LIN {X -0.176,Y -701.742,Z 1215.429,A 0.000,B 0.000,C 90.000,E1 113.259} C_DIS
LIN {X -0.039,Y -700.692,Z 1215.429,A 0.000,B 0.000,C 90.000,E1 113.131} C_DIS
LIN {X -0.019,Y -695.221,Z 1215.426,A 0.000,B 0.000,C 90.000,E1 112.695} C_DIS
LIN {X 0.002,Y -693.496,Z 1215.426,A 0.000,B 0.000,C 90.000,E1 112.589} C_DIS
LIN {X 0.017,Y -688.158,Z 1215.425,A 0.000,B 0.000,C 90.000,E1 112.408} C_DIS
LIN {X 0.322,Y -686.600,Z 1215.424,A 0.000,B 0.000,C 90.000,E1 112.333} C_DIS
LIN {X -0.036,Y -685.254,Z 1215.424,A 0.000,B 0.000,C 90.000,E1 112.333} C_DIS
LIN {X 0.238,Y -679.829,Z 1215.424,A 0.000,B 0.000,C 90.000,E1 112.280} C_DIS
LIN {X 0.132,Y -677.657,Z 1215.424,A 0.000,B 0.000,C 90.000,E1 112.280} C_DIS
LIN {X 0.079,Y -611.887,Z 1215.424,A 0.000,B 0.000,C 90.000,E1 112.280} C_DIS
LIN {X -0.103,Y -610.037,Z 1215.423,A 0.000,B 0.000,C 90.000,E1 112.206} C_DIS
LIN {X 0.141,Y -604.449,Z 1215.421,A 0.000,B 0.000,C 90.000,E1 111.791} C_DIS
LIN {X 0.099,Y -601.562,Z 1215.420,A 0.000,B 0.000,C 90.000,E1 111.535} C_DIS
LIN {X 0.143,Y -599.778,Z 1215.418,A 0.000,B 0.000,C 90.000,E1 111.280} C_DIS
LIN {X -0.112,Y -598.457,Z 1215.417,A 0.000,B 0.000,C 90.000,E1 111.153} C_DIS
LIN {X -0.155,Y -598.430,Z 1215.417,A 0.000,B 0.000,C 90.000,E1 111.153} C_DIS
LIN {X -0.070,Y -597.952,Z 1215.417,A 0.000,B 0.000,C 90.000,E1 110.972} C_DIS
LIN {X 0.221,Y -598.845,Z 1215.414,A 0.000,B 0.000,C 90.000,E1 110.482} C_DIS
LIN {X 0.094,Y -601.655,Z 1215.410,A 0.000,B 0.000,C 90.000,E1 109.704} C_DIS
LIN {X 0.200,Y -604.148,Z 1215.405,A 0.000,B 0.000,C 90.000,E1 108.906} C_DIS
LIN {X -0.243,Y -610.599,Z 1215.394,A 0.000,B 0.000,C 90.000,E1 106.858} C_DIS
LIN {X 0.087,Y -611.302,Z 1215.392,A 0.000,B 0.000,C 90.000,E1 106.567} C_DIS
LIN {X 0.007,Y -612.225,Z 1215.391,A 0.000,B 0.000,C 90.000,E1 106.315} C_DIS
LIN {X -0.145,Y -614.498,Z 1215.386,A 0.000,B 0.000,C 90.000,E1 105.552} C_DIS
LIN {X -0.108,Y -616.200,Z 1215.382,A 0.000,B 0.000,C 90.000,E1 104.773} C_DIS
LIN {X 0.020,Y -617.147,Z 1215.379,A 0.000,B 0.000,C 90.000,E1 104.245} C_DIS
LIN {X 0.159,Y -617.816,Z 1215.376,A 0.000,B 0.000,C 90.000,E1 103.716} C_DIS
LIN {X -0.157,Y -618.203,Z 1215.373,A 0.000,B 0.000,C 90.000,E1 103.231} C_DIS
LIN {X -0.014,Y -618.268,Z 1215.371,A 0.000,B 0.000,C 90.000,E1 102.703} C_DIS
LIN {X 0.360,Y -618.212,Z 1215.369,A 0.000,B 0.000,C 90.000,E1 102.411} C_DIS
LIN {X -0.229,Y -617.696,Z 1215.366,A 0.000,B 0.000,C 90.000,E1 101.951} C_DIS
LIN {X -0.083,Y -616.795,Z 1215.363,A 0.000,B 0.000,C 90.000,E1 101.422} C_DIS
LIN {X 0.054,Y -615.559,Z 1215.361,A 0.000,B 0.000,C 90.000,E1 100.894} C_DIS
LIN {X -0.184,Y -614.849,Z 1215.359,A 0.000,B 0.000,C 90.000,E1 100.658} C_DIS
LIN {X -0.172,Y -613.051,Z 1215.356,A 0.000,B 0.000,C 90.000,E1 100.141} C_DIS
LIN {X -0.242,Y -609.874,Z 1215.353,A 0.000,B 0.000,C 90.000,E1 99.500} C_DIS
LIN {X -0.077,Y -607.729,Z 1215.351,A 0.000,B 0.000,C 90.000,E1 99.095} C_DIS
LIN {X -0.198,Y -603.306,Z 1215.347,A 0.000,B 0.000,C 90.000,E1 98.454} C_DIS
LIN {X -0.254,Y -599.077,Z 1215.344,A 0.000,B 0.000,C 90.000,E1 97.936} C_DIS
LIN {X -0.212,Y -594.199,Z 1215.341,A 0.000,B 0.000,C 90.000,E1 97.409} C_DIS
LIN {X -0.018,Y -588.778,Z 1215.338,A 0.000,B 0.000,C 90.000,E1 96.891} C_DIS
LIN {X -0.118,Y -584.273,Z 1215.336,A 0.000,B 0.000,C 90.000,E1 96.543} C_DIS
LIN {X -0.046,Y -581.409,Z 1215.335,A 0.000,B 0.000,C 90.000,E1 96.315} C_DIS
LIN {X -0.022,Y -579.787,Z 1215.334,A 0.000,B 0.000,C 90.000,E1 96.201} C_DIS
LIN {X -0.082,Y -574.622,Z 1215.333,A 0.000,B 0.000,C 90.000,E1 95.910} C_DIS
LIN {X -0.113,Y -567.317,Z 1215.330,A 0.000,B 0.000,C 90.000,E1 95.454} C_DIS
LIN {X 0.093,Y -566.335,Z 1215.330,A 0.000,B 0.000,C 90.000,E1 95.334} C_DIS
LIN {X -0.087,Y -565.372,Z 1215.329,A 0.000,B 0.000,C 90.000,E1 95.220} C_DIS
LIN {X 0.152,Y -564.026,Z 1215.328,A 0.000,B 0.000,C 90.000,E1 94.935} C_DIS
LIN {X 0.109,Y -564.023,Z 1215.328,A 0.000,B 0.000,C 90.000,E1 94.935} C_DIS
LIN {X -0.143,Y -563.804,Z 1215.325,A 0.000,B 0.000,C 90.000,E1 94.531} C_DIS
LIN {X 0.187,Y -563.579,Z 1215.324,A 0.000,B 0.000,C 90.000,E1 94.359} C_DIS
LIN {X -0.278,Y -563.705,Z 1215.320,A 0.000,B 0.000,C 90.000,E1 93.555} C_DIS
LIN {X 0.274,Y -564.650,Z 1215.312,A 0.000,B 0.000,C 90.000,E1 92.121} C_DIS
LIN {X -0.062,Y -565.996,Z 1215.301,A 0.000,B 0.000,C 90.000,E1 90.229} C_DIS
LIN {X 0.068,Y -567.159,Z 1215.292,A 0.000,B 0.000,C 90.000,E1 88.568} C_DIS
LIN {X -0.007,Y -568.004,Z 1215.286,A 0.000,B 0.000,C 90.000,E1 87.478} C_DIS
LIN {X 0.210,Y -569.246,Z 1215.277,A 0.000,B 0.000,C 90.000,E1 85.812} C_DIS
LIN {X 0.060,Y -570.822,Z 1215.266,A 0.000,B 0.000,C 90.000,E1 83.913} C_DIS
LIN {X 0.201,Y -572.005,Z 1215.259,A 0.000,B 0.000,C 90.000,E1 82.534} C_DIS
LIN {X -0.060,Y -573.113,Z 1215.251,A 0.000,B 0.000,C 90.000,E1 81.197} C_DIS
LIN {X 0.274,Y -574.095,Z 1215.244,A 0.000,B 0.000,C 90.000,E1 79.803} C_DIS
LIN {X 0.259,Y -575.130,Z 1215.234,A 0.000,B 0.000,C 90.000,E1 78.173} C_DIS
LIN {X -0.189,Y -576.095,Z 1215.225,A 0.000,B 0.000,C 90.000,E1 76.589} C_DIS
LIN {X -0.132,Y -576.812,Z 1215.218,A 0.000,B 0.000,C 90.000,E1 75.227} C_DIS
LIN {X 0.303,Y -577.663,Z 1215.209,A 0.000,B 0.000,C 90.000,E1 73.559} C_DIS
LIN {X 0.223,Y -578.855,Z 1215.197,A 0.000,B 0.000,C 90.000,E1 71.402} C_DIS
LIN {X 0.002,Y -580.238,Z 1215.185,A 0.000,B 0.000,C 90.000,E1 69.263} C_DIS
LIN {X 0.067,Y -582.374,Z 1215.170,A 0.000,B 0.000,C 90.000,E1 66.561} C_DIS
LIN {X -0.194,Y -583.878,Z 1215.161,A 0.000,B 0.000,C 90.000,E1 64.973} C_DIS
LIN {X -0.014,Y -585.587,Z 1215.151,A 0.000,B 0.000,C 90.000,E1 63.076} C_DIS
LIN {X 0.054,Y -587.260,Z 1215.141,A 0.000,B 0.000,C 90.000,E1 61.463} C_DIS
LIN {X -0.073,Y -588.926,Z 1215.133,A 0.000,B 0.000,C 90.000,E1 59.871} C_DIS
LIN {X 0.147,Y -590.389,Z 1215.124,A 0.000,B 0.000,C 90.000,E1 58.250} C_DIS
LIN {X -0.005,Y -591.370,Z 1215.118,A 0.000,B 0.000,C 90.000,E1 57.199} C_DIS
LIN {X -0.002,Y -592.248,Z 1215.112,A 0.000,B 0.000,C 90.000,E1 56.135} C_DIS
LIN {X -0.218,Y -593.486,Z 1215.103,A 0.000,B 0.000,C 90.000,E1 54.562} C_DIS
LIN {X 0.269,Y -594.706,Z 1215.094,A 0.000,B 0.000,C 90.000,E1 52.924} C_DIS
LIN {X -0.141,Y -595.494,Z 1215.088,A 0.000,B 0.000,C 90.000,E1 51.904} C_DIS
LIN {X 0.290,Y -596.524,Z 1215.079,A 0.000,B 0.000,C 90.000,E1 50.275} C_DIS
LIN {X 0.285,Y -597.211,Z 1215.071,A 0.000,B 0.000,C 90.000,E1 48.690} C_DIS
LIN {X 0.064,Y -597.686,Z 1215.063,A 0.000,B 0.000,C 90.000,E1 47.391} C_DIS
LIN {X -0.156,Y -597.920,Z 1215.059,A 0.000,B 0.000,C 90.000,E1 46.620} C_DIS
LIN {X -0.179,Y -598.105,Z 1215.053,A 0.000,B 0.000,C 90.000,E1 45.567} C_DIS
LIN {X 0.019,Y -598.095,Z 1215.049,A 0.000,B 0.000,C 90.000,E1 44.757} C_DIS
LIN {X 0.217,Y -597.954,Z 1215.044,A 0.000,B 0.000,C 90.000,E1 43.947} C_DIS
LIN {X -0.217,Y -597.831,Z 1215.041,A 0.000,B 0.000,C 90.000,E1 43.461} C_DIS
LIN {X 0.186,Y -596.976,Z 1215.033,A 0.000,B 0.000,C 90.000,E1 41.838} C_DIS
LIN {X -0.040,Y -596.562,Z 1215.028,A 0.000,B 0.000,C 90.000,E1 41.067} C_DIS
LIN {X 0.175,Y -595.674,Z 1215.021,A 0.000,B 0.000,C 90.000,E1 39.725} C_DIS
LIN {X -0.072,Y -595.061,Z 1215.016,A 0.000,B 0.000,C 90.000,E1 38.955} C_DIS
LIN {X 0.208,Y -593.806,Z 1215.009,A 0.000,B 0.000,C 90.000,E1 37.604} C_DIS
LIN {X -0.216,Y -592.497,Z 1215.003,A 0.000,B 0.000,C 90.000,E1 36.583} C_DIS
LIN {X 0.215,Y -591.801,Z 1215.000,A 0.000,B 0.000,C 90.000,E1 36.011} C_DIS
LIN {X 0.100,Y -589.562,Z 1214.993,A 0.000,B 0.000,C 90.000,E1 34.692} C_DIS
LIN {X -0.115,Y -587.851,Z 1214.988,A 0.000,B 0.000,C 90.000,E1 33.913} C_DIS
LIN {X 0.138,Y -585.969,Z 1214.984,A 0.000,B 0.000,C 90.000,E1 33.086} C_DIS
LIN {X 0.187,Y -584.455,Z 1214.981,A 0.000,B 0.000,C 90.000,E1 32.546} C_DIS
LIN {X 0.258,Y -581.148,Z 1214.975,A 0.000,B 0.000,C 90.000,E1 31.465} C_DIS
LIN {X 0.130,Y -578.136,Z 1214.970,A 0.000,B 0.000,C 90.000,E1 30.669} C_DIS
LIN {X -0.016,Y -577.087,Z 1214.969,A 0.000,B 0.000,C 90.000,E1 30.413} C_DIS
LIN {X 0.024,Y -572.873,Z 1214.964,A 0.000,B 0.000,C 90.000,E1 29.461} C_DIS
LIN {X -0.303,Y -570.192,Z 1214.961,A 0.000,B 0.000,C 90.000,E1 28.949} C_DIS
LIN {X 0.215,Y -568.064,Z 1214.958,A 0.000,B 0.000,C 90.000,E1 28.487} C_DIS
LIN {X -0.231,Y -564.211,Z 1214.955,A 0.000,B 0.000,C 90.000,E1 27.847} C_DIS
LIN {X 0.151,Y -560.907,Z 1214.952,A 0.000,B 0.000,C 90.000,E1 27.257} C_DIS
LIN {X 0.045,Y -555.675,Z 1214.947,A 0.000,B 0.000,C 90.000,E1 26.437} C_DIS
LIN {X 0.242,Y -550.798,Z 1214.943,A 0.000,B 0.000,C 90.000,E1 25.720} C_DIS
LIN {X -0.221,Y -546.679,Z 1214.940,A 0.000,B 0.000,C 90.000,E1 25.207} C_DIS
LIN {X 0.149,Y -541.009,Z 1214.936,A 0.000,B 0.000,C 90.000,E1 24.463} C_DIS
LIN {X -0.020,Y -535.070,Z 1214.932,A 0.000,B 0.000,C 90.000,E1 23.770} C_DIS
LIN {X 0.160,Y -527.403,Z 1214.927,A 0.000,B 0.000,C 90.000,E1 22.898} C_DIS
LIN {X 0.124,Y -522.134,Z 1214.924,A 0.000,B 0.000,C 90.000,E1 22.333} C_DIS
LIN {X -0.185,Y -514.110,Z 1214.920,A 0.000,B 0.000,C 90.000,E1 21.535} C_DIS
LIN {X -0.222,Y -506.137,Z 1214.915,A 0.000,B 0.000,C 90.000,E1 20.737} C_DIS
LIN {X -0.144,Y -499.081,Z 1214.911,A 0.000,B 0.000,C 90.000,E1 20.047} C_DIS
LIN {X -0.219,Y -490.622,Z 1214.907,A 0.000,B 0.000,C 90.000,E1 19.268} C_DIS
LIN {X -0.006,Y -484.930,Z 1214.904,A 0.000,B 0.000,C 90.000,E1 18.725} C_DIS
LIN {X -0.059,Y -474.720,Z 1214.899,A 0.000,B 0.000,C 90.000,E1 17.819} C_DIS
LIN {X 0.239,Y -460.231,Z 1214.892,A 0.000,B 0.000,C 90.000,E1 16.496} C_DIS
LIN {X -0.140,Y -436.889,Z 1214.880,A 0.000,B 0.000,C 90.000,E1 14.356} C_DIS
LIN {X -0.031,Y -422.637,Z 1214.872,A 0.000,B 0.000,C 90.000,E1 12.883} C_DIS
LIN {X 0.152,Y -405.819,Z 1214.861,A 0.000,B 0.000,C 90.000,E1 10.950} C_DIS
LIN {X 0.016,Y -399.258,Z 1214.856,A 0.000,B 0.000,C 90.000,E1 10.141} C_DIS
LIN {X 0.006,Y -396.794,Z 1214.854,A 0.000,B 0.000,C 90.000,E1 9.792} C_DIS
LIN {X -0.168,Y -394.374,Z 1214.852,A 0.000,B 0.000,C 90.000,E1 9.378} C_DIS
LIN {X 0.140,Y -393.566,Z 1214.850,A 0.000,B 0.000,C 90.000,E1 9.029} C_DIS
LIN {X 0.103,Y -393.554,Z 1214.850,A 0.000,B 0.000,C 90.000,E1 9.029} C_DIS
LIN {X 0.109,Y -393.819,Z 1214.849,A 0.000,B 0.000,C 90.000,E1 8.746} C_DIS
LIN {X 0.071,Y -393.842,Z 1214.849,A 0.000,B 0.000,C 90.000,E1 8.746} C_DIS
LIN {X 0.065,Y -396.683,Z 1214.845,A 0.000,B 0.000,C 90.000,E1 8.106} C_DIS
LIN {X -0.154,Y -397.209,Z 1214.845,A 0.000,B 0.000,C 90.000,E1 8.049} C_DIS
LIN {X -0.152,Y -401.494,Z 1214.842,A 0.000,B 0.000,C 90.000,E1 7.530} C_DIS
LIN {X 0.103,Y -406.904,Z 1214.839,A 0.000,B 0.000,C 90.000,E1 7.011} C_DIS
LIN {X 0.092,Y -424.165,Z 1214.832,A 0.000,B 0.000,C 90.000,E1 5.682} C_DIS
LIN {X 0.068,Y -438.470,Z 1214.826,A 0.000,B 0.000,C 90.000,E1 4.588} C_DIS
LIN {X 0.149,Y -451.163,Z 1214.820,A 0.000,B 0.000,C 90.000,E1 3.612} C_DIS
LIN {X -0.098,Y -462.214,Z 1214.816,A 0.000,B 0.000,C 90.000,E1 2.808} C_DIS
LIN {X 0.170,Y -468.407,Z 1214.813,A 0.000,B 0.000,C 90.000,E1 2.293} C_DIS
LIN {X -0.127,Y -474.495,Z 1214.810,A 0.000,B 0.000,C 90.000,E1 1.835} C_DIS
LIN {X 0.089,Y -478.980,Z 1214.808,A 0.000,B 0.000,C 90.000,E1 1.432} C_DIS
LIN {X 0.032,Y -484.802,Z 1214.805,A 0.000,B 0.000,C 90.000,E1 0.917} C_DIS
LIN {X 0.169,Y -491.759,Z 1214.801,A 0.000,B 0.000,C 90.000,E1 0.229} C_DIS
LIN {X 0.215,Y -498.741,Z 1214.797,A 0.000,B 0.000,C 90.000,E1 359.484} C_DIS
LIN {X -0.234,Y -505.138,Z 1214.793,A 0.000,B 0.000,C 90.000,E1 358.797} C_DIS
LIN {X 0.101,Y -509.996,Z 1214.790,A 0.000,B 0.000,C 90.000,E1 358.165} C_DIS
LIN {X -0.158,Y -516.537,Z 1214.785,A 0.000,B 0.000,C 90.000,E1 357.306} C_DIS
LIN {X 0.250,Y -520.642,Z 1214.782,A 0.000,B 0.000,C 90.000,E1 356.674} C_DIS
LIN {X -0.147,Y -525.330,Z 1214.778,A 0.000,B 0.000,C 90.000,E1 355.988} C_DIS
LIN {X -0.193,Y -528.822,Z 1214.774,A 0.000,B 0.000,C 90.000,E1 355.412} C_DIS
LIN {X 0.041,Y -532.726,Z 1214.770,A 0.000,B 0.000,C 90.000,E1 354.666} C_DIS
LIN {X -0.166,Y -536.272,Z 1214.766,A 0.000,B 0.000,C 90.000,E1 353.970} C_DIS
LIN {X -0.126,Y -538.907,Z 1214.763,A 0.000,B 0.000,C 90.000,E1 353.394} C_DIS
LIN {X 0.001,Y -543.614,Z 1214.757,A 0.000,B 0.000,C 90.000,E1 352.243} C_DIS
LIN {X 0.169,Y -546.694,Z 1214.752,A 0.000,B 0.000,C 90.000,E1 351.376} C_DIS
LIN {X -0.071,Y -550.337,Z 1214.746,A 0.000,B 0.000,C 90.000,E1 350.274} C_DIS
LIN {X -0.164,Y -553.559,Z 1214.740,A 0.000,B 0.000,C 90.000,E1 349.162} C_DIS
LIN {X -0.070,Y -557.218,Z 1214.732,A 0.000,B 0.000,C 90.000,E1 347.757} C_DIS
LIN {X -0.201,Y -559.175,Z 1214.727,A 0.000,B 0.000,C 90.000,E1 346.937} C_DIS
LIN {X -0.316,Y -561.054,Z 1214.723,A 0.000,B 0.000,C 90.000,E1 346.117} C_DIS
LIN {X 0.028,Y -563.906,Z 1214.715,A 0.000,B 0.000,C 90.000,E1 344.700} C_DIS
LIN {X 0.029,Y -566.515,Z 1214.707,A 0.000,B 0.000,C 90.000,E1 343.323} C_DIS
LIN {X -0.080,Y -568.342,Z 1214.701,A 0.000,B 0.000,C 90.000,E1 342.236} C_DIS
LIN {X -0.161,Y -569.994,Z 1214.695,A 0.000,B 0.000,C 90.000,E1 341.148} C_DIS
LIN {X -0.221,Y -571.395,Z 1214.689,A 0.000,B 0.000,C 90.000,E1 340.061} C_DIS
LIN {X -0.068,Y -572.466,Z 1214.683,A 0.000,B 0.000,C 90.000,E1 338.954} C_DIS
LIN {X 0.271,Y -573.013,Z 1214.679,A 0.000,B 0.000,C 90.000,E1 338.103} C_DIS
LIN {X -0.089,Y -573.246,Z 1214.672,A 0.000,B 0.000,C 90.000,E1 337.050} C_DIS
LIN {X -0.056,Y -573.101,Z 1214.668,A 0.000,B 0.000,C 90.000,E1 336.230} C_DIS
LIN {X -0.181,Y -572.418,Z 1214.662,A 0.000,B 0.000,C 90.000,E1 335.153} C_DIS
LIN {X 0.201,Y -571.062,Z 1214.656,A 0.000,B 0.000,C 90.000,E1 334.024} C_DIS
LIN {X -0.132,Y -570.113,Z 1214.653,A 0.000,B 0.000,C 90.000,E1 333.512} C_DIS
LIN {X -0.049,Y -567.696,Z 1214.647,A 0.000,B 0.000,C 90.000,E1 332.410} C_DIS
LIN {X -0.084,Y -565.580,Z 1214.642,A 0.000,B 0.000,C 90.000,E1 331.591} C_DIS
LIN {X 0.118,Y -562.896,Z 1214.638,A 0.000,B 0.000,C 90.000,E1 330.745} C_DIS
LIN {X 0.082,Y -559.403,Z 1214.633,A 0.000,B 0.000,C 90.000,E1 329.921} C_DIS
LIN {X -0.333,Y -556.642,Z 1214.630,A 0.000,B 0.000,C 90.000,E1 329.410} C_DIS
LIN {X 0.160,Y -552.750,Z 1214.626,A 0.000,B 0.000,C 90.000,E1 328.663} C_DIS
LIN {X -0.263,Y -547.301,Z 1214.621,A 0.000,B 0.000,C 90.000,E1 327.867} C_DIS
LIN {X 0.272,Y -543.238,Z 1214.618,A 0.000,B 0.000,C 90.000,E1 327.248} C_DIS
LIN {X 0.025,Y -539.006,Z 1214.615,A 0.000,B 0.000,C 90.000,E1 326.707} C_DIS
LIN {X -0.097,Y -533.297,Z 1214.611,A 0.000,B 0.000,C 90.000,E1 326.008} C_DIS
LIN {X -0.104,Y -519.243,Z 1214.602,A 0.000,B 0.000,C 90.000,E1 324.276} C_DIS
LIN {X 0.007,Y -515.632,Z 1214.599,A 0.000,B 0.000,C 90.000,E1 323.749} C_DIS
LIN {X -0.093,Y -512.750,Z 1214.596,A 0.000,B 0.000,C 90.000,E1 323.256} C_DIS
LIN {X 0.088,Y -510.843,Z 1214.593,A 0.000,B 0.000,C 90.000,E1 322.763} C_DIS
LIN {X 0.008,Y -510.074,Z 1214.592,A 0.000,B 0.000,C 90.000,E1 322.477} C_DIS
LIN {X -0.167,Y -509.170,Z 1214.588,A 0.000,B 0.000,C 90.000,E1 321.904} C_DIS
LIN {X -0.203,Y -508.932,Z 1214.587,A 0.000,B 0.000,C 90.000,E1 321.618} C_DIS
LIN {X -0.162,Y -508.760,Z 1214.582,A 0.000,B 0.000,C 90.000,E1 320.723} C_DIS
LIN {X 0.201,Y -510.310,Z 1214.565,A 0.000,B 0.000,C 90.000,E1 317.715} C_DIS
LIN {X 0.146,Y -511.522,Z 1214.554,A 0.000,B 0.000,C 90.000,E1 315.648} C_DIS
LIN {X -0.286,Y -512.148,Z 1214.547,A 0.000,B 0.000,C 90.000,E1 314.514} C_DIS
LIN {X 0.084,Y -513.159,Z 1214.536,A 0.000,B 0.000,C 90.000,E1 312.405} C_DIS
LIN {X -0.037,Y -513.925,Z 1214.527,A 0.000,B 0.000,C 90.000,E1 310.943} C_DIS
LIN {X -0.154,Y -514.655,Z 1214.519,A 0.000,B 0.000,C 90.000,E1 309.483} C_DIS
LIN {X -0.053,Y -515.004,Z 1214.514,A 0.000,B 0.000,C 90.000,E1 308.588} C_DIS
LIN {X 0.071,Y -515.402,Z 1214.508,A 0.000,B 0.000,C 90.000,E1 307.397} C_DIS
LIN {X 0.038,Y -515.983,Z 1214.500,A 0.000,B 0.000,C 90.000,E1 305.931} C_DIS
LIN {X -0.242,Y -516.762,Z 1214.490,A 0.000,B 0.000,C 90.000,E1 304.199} C_DIS
LIN {X -0.001,Y -517.295,Z 1214.482,A 0.000,B 0.000,C 90.000,E1 302.704} C_DIS
LIN {X -0.190,Y -517.754,Z 1214.474,A 0.000,B 0.000,C 90.000,E1 301.258} C_DIS
LIN {X -0.130,Y -517.944,Z 1214.467,A 0.000,B 0.000,C 90.000,E1 300.079} C_DIS
LIN {X -0.021,Y -518.189,Z 1214.457,A 0.000,B 0.000,C 90.000,E1 298.309} C_DIS
LIN {X 0.080,Y -518.389,Z 1214.448,A 0.000,B 0.000,C 90.000,E1 296.539} C_DIS
LIN {X -0.156,Y -518.442,Z 1214.436,A 0.000,B 0.000,C 90.000,E1 294.515} C_DIS
LIN {X -0.266,Y -518.508,Z 1214.426,A 0.000,B 0.000,C 90.000,E1 292.770} C_DIS
LIN {X -0.038,Y -518.509,Z 1214.418,A 0.000,B 0.000,C 90.000,E1 291.280} C_DIS
LIN {X -0.004,Y -517.983,Z 1214.410,A 0.000,B 0.000,C 90.000,E1 289.812} C_DIS
LIN {X -0.121,Y -517.512,Z 1214.404,A 0.000,B 0.000,C 90.000,E1 288.652} C_DIS
LIN {X 0.182,Y -516.592,Z 1214.394,A 0.000,B 0.000,C 90.000,E1 286.858} C_DIS
LIN {X -0.239,Y -516.101,Z 1214.389,A 0.000,B 0.000,C 90.000,E1 286.024} C_DIS
LIN {X 0.004,Y -514.821,Z 1214.377,A 0.000,B 0.000,C 90.000,E1 283.939} C_DIS
LIN {X -0.106,Y -513.925,Z 1214.369,A 0.000,B 0.000,C 90.000,E1 282.479} C_DIS
LIN {X -0.121,Y -512.918,Z 1214.361,A 0.000,B 0.000,C 90.000,E1 281.007} C_DIS
LIN {X 0.120,Y -511.853,Z 1214.351,A 0.000,B 0.000,C 90.000,E1 279.208} C_DIS
LIN {X 0.231,Y -510.509,Z 1214.340,A 0.000,B 0.000,C 90.000,E1 277.125} C_DIS
LIN {X -0.161,Y -509.518,Z 1214.330,A 0.000,B 0.000,C 90.000,E1 275.391} C_DIS
LIN {X -0.167,Y -508.483,Z 1214.320,A 0.000,B 0.000,C 90.000,E1 273.612} C_DIS
LIN {X 0.111,Y -507.062,Z 1214.307,A 0.000,B 0.000,C 90.000,E1 271.203} C_DIS
LIN {X 0.121,Y -506.158,Z 1214.299,A 0.000,B 0.000,C 90.000,E1 269.714} C_DIS
LIN {X 0.216,Y -505.540,Z 1214.292,A 0.000,B 0.000,C 90.000,E1 268.511} C_DIS
LIN {X 0.122,Y -504.449,Z 1214.282,A 0.000,B 0.000,C 90.000,E1 266.731} C_DIS
LIN {X 0.087,Y -503.466,Z 1214.274,A 0.000,B 0.000,C 90.000,E1 265.241} C_DIS
LIN {X 0.041,Y -502.072,Z 1214.264,A 0.000,B 0.000,C 90.000,E1 263.451} C_DIS
LIN {X 0.047,Y -500.650,Z 1214.255,A 0.000,B 0.000,C 90.000,E1 261.951} C_DIS
LIN {X 0.094,Y -499.304,Z 1214.247,A 0.000,B 0.000,C 90.000,E1 260.443} C_DIS
LIN {X 0.043,Y -497.586,Z 1214.235,A 0.000,B 0.000,C 90.000,E1 258.342} C_DIS
LIN {X 0.051,Y -495.982,Z 1214.224,A 0.000,B 0.000,C 90.000,E1 256.228} C_DIS
LIN {X 0.123,Y -494.452,Z 1214.212,A 0.000,B 0.000,C 90.000,E1 254.102} C_DIS
LIN {X -0.129,Y -492.951,Z 1214.197,A 0.000,B 0.000,C 90.000,E1 251.402} C_DIS
LIN {X -0.136,Y -492.356,Z 1214.190,A 0.000,B 0.000,C 90.000,E1 250.188} C_DIS
LIN {X 0.060,Y -491.440,Z 1214.181,A 0.000,B 0.000,C 90.000,E1 248.646} C_DIS
LIN {X 0.241,Y -490.345,Z 1214.173,A 0.000,B 0.000,C 90.000,E1 247.102} C_DIS
LIN {X -0.085,Y -489.237,Z 1214.166,A 0.000,B 0.000,C 90.000,E1 245.921} C_DIS
LIN {X -0.208,Y -487.724,Z 1214.158,A 0.000,B 0.000,C 90.000,E1 244.409} C_DIS
LIN {X -0.147,Y -486.136,Z 1214.149,A 0.000,B 0.000,C 90.000,E1 242.871} C_DIS
LIN {X -0.103,Y -483.582,Z 1214.137,A 0.000,B 0.000,C 90.000,E1 240.717} C_DIS
LIN {X 0.123,Y -482.104,Z 1214.130,A 0.000,B 0.000,C 90.000,E1 239.459} C_DIS
LIN {X 0.124,Y -480.203,Z 1214.122,A 0.000,B 0.000,C 90.000,E1 237.916} C_DIS
LIN {X 0.076,Y -477.661,Z 1214.110,A 0.000,B 0.000,C 90.000,E1 235.754} C_DIS
LIN {X 0.089,Y -475.192,Z 1214.098,A 0.000,B 0.000,C 90.000,E1 233.577} C_DIS
LIN {X -0.005,Y -473.465,Z 1214.089,A 0.000,B 0.000,C 90.000,E1 232.029} C_DIS
LIN {X 0.104,Y -471.262,Z 1214.077,A 0.000,B 0.000,C 90.000,E1 229.828} C_DIS
LIN {X 0.008,Y -469.432,Z 1214.067,A 0.000,B 0.000,C 90.000,E1 227.957} C_DIS
LIN {X 0.074,Y -467.890,Z 1214.058,A 0.000,B 0.000,C 90.000,E1 226.377} C_DIS
LIN {X -0.079,Y -465.980,Z 1214.046,A 0.000,B 0.000,C 90.000,E1 224.190} C_DIS
LIN {X 0.056,Y -464.181,Z 1214.024,A 0.000,B 0.000,C 90.000,E1 220.378} C_DIS
LIN {X -0.239,Y -464.727,Z 1214.002,A 0.000,B 0.000,C 90.000,E1 216.297} C_DIS
LIN {X -0.293,Y -465.368,Z 1213.991,A 0.000,B 0.000,C 90.000,E1 214.405} C_DIS
LIN {X -0.097,Y -466.268,Z 1213.982,A 0.000,B 0.000,C 90.000,E1 212.801} C_DIS
LIN {X 0.165,Y -467.966,Z 1213.972,A 0.000,B 0.000,C 90.000,E1 210.875} C_DIS
LIN {X 0.164,Y -470.563,Z 1213.958,A 0.000,B 0.000,C 90.000,E1 208.359} C_DIS
LIN {X -0.084,Y -472.457,Z 1213.949,A 0.000,B 0.000,C 90.000,E1 206.821} C_DIS
LIN {X 0.207,Y -473.513,Z 1213.944,A 0.000,B 0.000,C 90.000,E1 205.848} C_DIS
LIN {X -0.295,Y -474.379,Z 1213.940,A 0.000,B 0.000,C 90.000,E1 205.283} C_DIS
LIN {X -0.097,Y -477.355,Z 1213.928,A 0.000,B 0.000,C 90.000,E1 203.078} C_DIS
LIN {X 0.098,Y -484.703,Z 1213.906,A 0.000,B 0.000,C 90.000,E1 199.033} C_DIS
LIN {X -0.145,Y -488.794,Z 1213.896,A 0.000,B 0.000,C 90.000,E1 197.221} C_DIS
LIN {X -0.054,Y -494.848,Z 1213.882,A 0.000,B 0.000,C 90.000,E1 194.773} C_DIS
LIN {X 0.044,Y -500.719,Z 1213.870,A 0.000,B 0.000,C 90.000,E1 192.647} C_DIS
LIN {X -0.237,Y -504.213,Z 1213.864,A 0.000,B 0.000,C 90.000,E1 191.478} C_DIS
LIN {X 0.196,Y -512.987,Z 1213.847,A 0.000,B 0.000,C 90.000,E1 188.454} C_DIS
LIN {X -0.018,Y -517.591,Z 1213.839,A 0.000,B 0.000,C 90.000,E1 187.004} C_DIS
LIN {X -0.209,Y -521.202,Z 1213.832,A 0.000,B 0.000,C 90.000,E1 185.853} C_DIS
LIN {X 0.084,Y -526.449,Z 1213.823,A 0.000,B 0.000,C 90.000,E1 184.073} C_DIS
LIN {X 0.018,Y -529.976,Z 1213.816,A 0.000,B 0.000,C 90.000,E1 182.922} C_DIS
LIN {X -0.034,Y -533.490,Z 1213.810,A 0.000,B 0.000,C 90.000,E1 181.776} C_DIS
LIN {X -0.044,Y -537.912,Z 1213.802,A 0.000,B 0.000,C 90.000,E1 180.344} C_DIS
LIN {X -0.009,Y -540.562,Z 1213.797,A 0.000,B 0.000,C 90.000,E1 179.484} C_DIS
LIN {X 0.159,Y -545.648,Z 1213.788,A 0.000,B 0.000,C 90.000,E1 177.764} C_DIS
LIN {X -0.114,Y -550.574,Z 1213.778,A 0.000,B 0.000,C 90.000,E1 176.102} C_DIS
LIN {X -0.209,Y -555.294,Z 1213.769,A 0.000,B 0.000,C 90.000,E1 174.432} C_DIS
LIN {X 0.157,Y -558.382,Z 1213.763,A 0.000,B 0.000,C 90.000,E1 173.280} C_DIS
LIN {X -0.183,Y -563.634,Z 1213.752,A 0.000,B 0.000,C 90.000,E1 171.376} C_DIS
LIN {X -0.018,Y -567.362,Z 1213.744,A 0.000,B 0.000,C 90.000,E1 169.982} C_DIS
LIN {X -0.048,Y -571.768,Z 1213.735,A 0.000,B 0.000,C 90.000,E1 168.342} C_DIS
LIN {X -0.024,Y -574.004,Z 1213.731,A 0.000,B 0.000,C 90.000,E1 167.521} C_DIS
LIN {X -0.261,Y -579.291,Z 1213.720,A 0.000,B 0.000,C 90.000,E1 165.644} C_DIS
LIN {X 0.246,Y -583.994,Z 1213.711,A 0.000,B 0.000,C 90.000,E1 163.976} C_DIS
LIN {X 0.299,Y -588.834,Z 1213.702,A 0.000,B 0.000,C 90.000,E1 162.362} C_DIS
LIN {X 0.252,Y -598.299,Z 1213.686,A 0.000,B 0.000,C 90.000,E1 159.444} C_DIS
LIN {X -0.126,Y -603.972,Z 1213.677,A 0.000,B 0.000,C 90.000,E1 157.901} C_DIS
LIN {X -0.347,Y -608.657,Z 1213.670,A 0.000,B 0.000,C 90.000,E1 156.613} C_DIS
LIN {X -0.005,Y -613.266,Z 1213.663,A 0.000,B 0.000,C 90.000,E1 155.281} C_DIS
LIN {X 0.178,Y -616.832,Z 1213.657,A 0.000,B 0.000,C 90.000,E1 154.229} C_DIS
LIN {X 0.114,Y -620.276,Z 1213.651,A 0.000,B 0.000,C 90.000,E1 153.204} C_DIS
LIN {X 0.385,Y -623.562,Z 1213.646,A 0.000,B 0.000,C 90.000,E1 152.153} C_DIS
LIN {X -0.111,Y -628.421,Z 1213.637,A 0.000,B 0.000,C 90.000,E1 150.667} C_DIS
LIN {X 0.104,Y -633.107,Z 1213.629,A 0.000,B 0.000,C 90.000,E1 149.125} C_DIS
LIN {X 0.016,Y -636.143,Z 1213.623,A 0.000,B 0.000,C 90.000,E1 148.122} C_DIS
LIN {X 0.347,Y -639.753,Z 1213.616,A 0.000,B 0.000,C 90.000,E1 146.834} C_DIS
LIN {X 0.201,Y -643.060,Z 1213.609,A 0.000,B 0.000,C 90.000,E1 145.595} C_DIS
LIN {X 0.101,Y -646.185,Z 1213.602,A 0.000,B 0.000,C 90.000,E1 144.356} C_DIS
LIN {X -0.011,Y -648.400,Z 1213.597,A 0.000,B 0.000,C 90.000,E1 143.371} C_DIS
LIN {X -0.251,Y -651.663,Z 1213.588,A 0.000,B 0.000,C 90.000,E1 141.904} C_DIS
LIN {X 0.049,Y -654.332,Z 1213.581,A 0.000,B 0.000,C 90.000,E1 140.642} C_DIS
LIN {X -0.072,Y -657.468,Z 1213.573,A 0.000,B 0.000,C 90.000,E1 139.175} C_DIS
LIN {X -0.233,Y -661.205,Z 1213.564,A 0.000,B 0.000,C 90.000,E1 137.472} C_DIS
LIN {X 0.148,Y -664.868,Z 1213.554,A 0.000,B 0.000,C 90.000,E1 135.729} C_DIS
LIN {X 0.147,Y -669.411,Z 1213.543,A 0.000,B 0.000,C 90.000,E1 133.785} C_DIS
LIN {X 0.270,Y -673.652,Z 1213.534,A 0.000,B 0.000,C 90.000,E1 132.081} C_DIS
LIN {X 0.046,Y -677.782,Z 1213.525,A 0.000,B 0.000,C 90.000,E1 130.415} C_DIS
LIN {X -0.124,Y -681.371,Z 1213.517,A 0.000,B 0.000,C 90.000,E1 128.991} C_DIS
LIN {X 0.301,Y -684.923,Z 1213.509,A 0.000,B 0.000,C 90.000,E1 127.523} C_DIS
LIN {X -0.181,Y -688.549,Z 1213.501,A 0.000,B 0.000,C 90.000,E1 126.137} C_DIS
LIN {X 0.112,Y -691.821,Z 1213.493,A 0.000,B 0.000,C 90.000,E1 124.692} C_DIS
LIN {X -0.351,Y -693.977,Z 1213.488,A 0.000,B 0.000,C 90.000,E1 123.785} C_DIS
LIN {X 0.405,Y -696.630,Z 1213.481,A 0.000,B 0.000,C 90.000,E1 122.546} C_DIS
LIN {X -0.384,Y -698.558,Z 1213.476,A 0.000,B 0.000,C 90.000,E1 121.671} C_DIS
LIN {X 0.071,Y -700.826,Z 1213.469,A 0.000,B 0.000,C 90.000,E1 120.463} C_DIS
LIN {X 0.210,Y -703.018,Z 1213.463,A 0.000,B 0.000,C 90.000,E1 119.283} C_DIS
LIN {X 0.101,Y -704.538,Z 1213.458,A 0.000,B 0.000,C 90.000,E1 118.359} C_DIS
LIN {X 0.338,Y -705.464,Z 1213.454,A 0.000,B 0.000,C 90.000,E1 117.641} C_DIS
LIN {X -0.033,Y -705.908,Z 1213.451,A 0.000,B 0.000,C 90.000,E1 117.206} C_DIS
LIN {X 0.217,Y -706.346,Z 1213.447,A 0.000,B 0.000,C 90.000,E1 116.488} C_DIS
LIN {X 0.155,Y -706.674,Z 1213.443,A 0.000,B 0.000,C 90.000,E1 115.796} C_DIS
LIN {X 0.100,Y -706.619,Z 1213.440,A 0.000,B 0.000,C 90.000,E1 115.103} C_DIS
LIN {X 0.049,Y -706.311,Z 1213.437,A 0.000,B 0.000,C 90.000,E1 114.643} C_DIS
LIN {X 0.340,Y -706.016,Z 1213.436,A 0.000,B 0.000,C 90.000,E1 114.387} C_DIS
LIN {X -0.014,Y -705.137,Z 1213.433,A 0.000,B 0.000,C 90.000,E1 113.951} C_DIS
LIN {X 0.273,Y -704.166,Z 1213.432,A 0.000,B 0.000,C 90.000,E1 113.695} C_DIS
LIN {X -0.089,Y -701.830,Z 1213.429,A 0.000,B 0.000,C 90.000,E1 113.259} C_DIS
LIN {X 0.049,Y -700.808,Z 1213.429,A 0.000,B 0.000,C 90.000,E1 113.131} C_DIS
LIN {X 0.061,Y -695.334,Z 1213.426,A 0.000,B 0.000,C 90.000,E1 112.695} C_DIS
LIN {X 0.082,Y -693.665,Z 1213.426,A 0.000,B 0.000,C 90.000,E1 112.589} C_DIS
LIN {X -0.121,Y -691.162,Z 1213.425,A 0.000,B 0.000,C 90.000,E1 112.514} C_DIS
LIN {X 0.321,Y -686.709,Z 1213.424,A 0.000,B 0.000,C 90.000,E1 112.333} C_DIS
LIN {X 0.008,Y -685.663,Z 1213.424,A 0.000,B 0.000,C 90.000,E1 112.333} C_DIS
LIN {X 0.222,Y -680.045,Z 1213.424,A 0.000,B 0.000,C 90.000,E1 112.280} C_DIS
LIN {X 0.115,Y -677.873,Z 1213.424,A 0.000,B 0.000,C 90.000,E1 112.280} C_DIS
LIN {X 0.064,Y -611.258,Z 1213.424,A 0.000,B 0.000,C 90.000,E1 112.280} C_DIS
LIN {X -0.117,Y -609.401,Z 1213.423,A 0.000,B 0.000,C 90.000,E1 112.206} C_DIS
LIN {X 0.179,Y -603.865,Z 1213.421,A 0.000,B 0.000,C 90.000,E1 111.791} C_DIS
LIN {X 0.143,Y -600.847,Z 1213.420,A 0.000,B 0.000,C 90.000,E1 111.535} C_DIS
LIN {X 0.260,Y -599.956,Z 1213.419,A 0.000,B 0.000,C 90.000,E1 111.408} C_DIS
LIN {X 0.098,Y -597.390,Z 1213.418,A 0.000,B 0.000,C 90.000,E1 111.153} C_DIS
LIN {X -0.035,Y -595.953,Z 1213.416,A 0.000,B 0.000,C 90.000,E1 110.865} C_DIS
LIN {X -0.078,Y -595.956,Z 1213.416,A 0.000,B 0.000,C 90.000,E1 110.865} C_DIS
LIN {X 0.204,Y -596.571,Z 1213.414,A 0.000,B 0.000,C 90.000,E1 110.482} C_DIS
LIN {X -0.105,Y -597.280,Z 1213.412,A 0.000,B 0.000,C 90.000,E1 110.248} C_DIS
LIN {X -0.313,Y -600.877,Z 1213.407,A 0.000,B 0.000,C 90.000,E1 109.214} C_DIS
LIN {X -0.221,Y -603.223,Z 1213.402,A 0.000,B 0.000,C 90.000,E1 108.417} C_DIS
LIN {X 0.187,Y -606.219,Z 1213.396,A 0.000,B 0.000,C 90.000,E1 107.330} C_DIS
LIN {X -0.032,Y -608.591,Z 1213.392,A 0.000,B 0.000,C 90.000,E1 106.567} C_DIS
LIN {X -0.050,Y -610.776,Z 1213.388,A 0.000,B 0.000,C 90.000,E1 105.788} C_DIS
LIN {X -0.051,Y -612.451,Z 1213.383,A 0.000,B 0.000,C 90.000,E1 105.009} C_DIS
LIN {X 0.050,Y -613.394,Z 1213.380,A 0.000,B 0.000,C 90.000,E1 104.481} C_DIS
LIN {X 0.067,Y -614.331,Z 1213.376,A 0.000,B 0.000,C 90.000,E1 103.703} C_DIS
LIN {X 0.183,Y -614.610,Z 1213.373,A 0.000,B 0.000,C 90.000,E1 103.175} C_DIS
LIN {X 0.301,Y -614.530,Z 1213.370,A 0.000,B 0.000,C 90.000,E1 102.647} C_DIS
LIN {X -0.179,Y -614.081,Z 1213.368,A 0.000,B 0.000,C 90.000,E1 102.175} C_DIS
LIN {X 0.179,Y -613.748,Z 1213.366,A 0.000,B 0.000,C 90.000,E1 101.883} C_DIS
LIN {X 0.171,Y -612.717,Z 1213.363,A 0.000,B 0.000,C 90.000,E1 101.366} C_DIS
LIN {X 0.280,Y -611.381,Z 1213.360,A 0.000,B 0.000,C 90.000,E1 100.838} C_DIS
LIN {X -0.223,Y -609.522,Z 1213.358,A 0.000,B 0.000,C 90.000,E1 100.366} C_DIS
LIN {X 0.272,Y -606.472,Z 1213.354,A 0.000,B 0.000,C 90.000,E1 99.670} C_DIS
LIN {X 0.138,Y -602.492,Z 1213.350,A 0.000,B 0.000,C 90.000,E1 99.029} C_DIS
LIN {X 0.069,Y -598.825,Z 1213.347,A 0.000,B 0.000,C 90.000,E1 98.511} C_DIS
LIN {X -0.020,Y -594.545,Z 1213.344,A 0.000,B 0.000,C 90.000,E1 97.992} C_DIS
LIN {X -0.031,Y -589.652,Z 1213.342,A 0.000,B 0.000,C 90.000,E1 97.466} C_DIS
LIN {X 0.075,Y -585.298,Z 1213.339,A 0.000,B 0.000,C 90.000,E1 97.068} C_DIS
LIN {X -0.019,Y -580.884,Z 1213.337,A 0.000,B 0.000,C 90.000,E1 96.720} C_DIS
LIN {X 0.113,Y -577.635,Z 1213.336,A 0.000,B 0.000,C 90.000,E1 96.486} C_DIS
LIN {X 0.011,Y -572.873,Z 1213.334,A 0.000,B 0.000,C 90.000,E1 96.201} C_DIS
LIN {X -0.167,Y -568.537,Z 1213.333,A 0.000,B 0.000,C 90.000,E1 95.910} C_DIS
LIN {X -0.098,Y -567.277,Z 1213.332,A 0.000,B 0.000,C 90.000,E1 95.796} C_DIS
LIN {X 0.131,Y -564.045,Z 1213.330,A 0.000,B 0.000,C 90.000,E1 95.391} C_DIS
LIN {X -0.100,Y -563.576,Z 1213.329,A 0.000,B 0.000,C 90.000,E1 95.277} C_DIS
LIN {X -0.091,Y -563.291,Z 1213.325,A 0.000,B 0.000,C 90.000,E1 94.588} C_DIS
LIN {X -0.118,Y -563.748,Z 1213.318,A 0.000,B 0.000,C 90.000,E1 93.212} C_DIS
LIN {X 0.224,Y -564.389,Z 1213.313,A 0.000,B 0.000,C 90.000,E1 92.350} C_DIS
LIN {X 0.221,Y -565.351,Z 1213.306,A 0.000,B 0.000,C 90.000,E1 90.974} C_DIS
LIN {X 0.224,Y -566.354,Z 1213.298,A 0.000,B 0.000,C 90.000,E1 89.599} C_DIS
LIN {X 0.048,Y -567.990,Z 1213.286,A 0.000,B 0.000,C 90.000,E1 87.421} C_DIS
LIN {X 0.265,Y -569.220,Z 1213.277,A 0.000,B 0.000,C 90.000,E1 85.755} C_DIS
LIN {X 0.113,Y -570.782,Z 1213.266,A 0.000,B 0.000,C 90.000,E1 83.856} C_DIS
LIN {X -0.243,Y -571.939,Z 1213.258,A 0.000,B 0.000,C 90.000,E1 82.527} C_DIS
LIN {X -0.014,Y -573.033,Z 1213.251,A 0.000,B 0.000,C 90.000,E1 81.141} C_DIS
LIN {X -0.248,Y -573.989,Z 1213.243,A 0.000,B 0.000,C 90.000,E1 79.803} C_DIS
LIN {X -0.266,Y -575.023,Z 1213.234,A 0.000,B 0.000,C 90.000,E1 78.173} C_DIS
LIN {X 0.185,Y -576.110,Z 1213.224,A 0.000,B 0.000,C 90.000,E1 76.228} C_DIS
LIN {X 0.250,Y -576.796,Z 1213.216,A 0.000,B 0.000,C 90.000,E1 74.866} C_DIS
LIN {X -0.233,Y -577.524,Z 1213.209,A 0.000,B 0.000,C 90.000,E1 73.559} C_DIS
LIN {X 0.036,Y -578.584,Z 1213.198,A 0.000,B 0.000,C 90.000,E1 71.638} C_DIS
LIN {X 0.124,Y -579.532,Z 1213.189,A 0.000,B 0.000,C 90.000,E1 70.007} C_DIS
LIN {X -0.119,Y -580.687,Z 1213.180,A 0.000,B 0.000,C 90.000,E1 68.411} C_DIS
LIN {X 0.282,Y -582.266,Z 1213.170,A 0.000,B 0.000,C 90.000,E1 66.485} C_DIS
LIN {X -0.089,Y -583.538,Z 1213.162,A 0.000,B 0.000,C 90.000,E1 65.177} C_DIS
LIN {X -0.186,Y -585.269,Z 1213.152,A 0.000,B 0.000,C 90.000,E1 63.307} C_DIS
LIN {X -0.227,Y -587.180,Z 1213.141,A 0.000,B 0.000,C 90.000,E1 61.435} C_DIS
LIN {X -0.011,Y -588.569,Z 1213.134,A 0.000,B 0.000,C 90.000,E1 60.078} C_DIS
LIN {X 0.006,Y -589.819,Z 1213.126,A 0.000,B 0.000,C 90.000,E1 58.742} C_DIS
LIN {X 0.041,Y -591.040,Z 1213.119,A 0.000,B 0.000,C 90.000,E1 57.406} C_DIS
LIN {X -0.083,Y -592.111,Z 1213.112,A 0.000,B 0.000,C 90.000,E1 56.087} C_DIS
LIN {X 0.033,Y -593.344,Z 1213.103,A 0.000,B 0.000,C 90.000,E1 54.482} C_DIS
LIN {X -0.311,Y -594.571,Z 1213.094,A 0.000,B 0.000,C 90.000,E1 52.924} C_DIS
LIN {X 0.112,Y -595.335,Z 1213.088,A 0.000,B 0.000,C 90.000,E1 51.823} C_DIS
LIN {X -0.298,Y -596.367,Z 1213.079,A 0.000,B 0.000,C 90.000,E1 50.275} C_DIS
LIN {X -0.081,Y -596.943,Z 1213.072,A 0.000,B 0.000,C 90.000,E1 48.933} C_DIS
LIN {X -0.308,Y -597.436,Z 1213.065,A 0.000,B 0.000,C 90.000,E1 47.634} C_DIS
LIN {X 0.092,Y -597.730,Z 1213.059,A 0.000,B 0.000,C 90.000,E1 46.539} C_DIS
LIN {X -0.149,Y -597.936,Z 1213.051,A 0.000,B 0.000,C 90.000,E1 45.243} C_DIS
LIN {X -0.387,Y -597.722,Z 1213.044,A 0.000,B 0.000,C 90.000,E1 43.947} C_DIS
LIN {X -0.197,Y -597.448,Z 1213.040,A 0.000,B 0.000,C 90.000,E1 43.137} C_DIS
LIN {X -0.025,Y -596.722,Z 1213.032,A 0.000,B 0.000,C 90.000,E1 41.800} C_DIS
LIN {X 0.191,Y -596.291,Z 1213.028,A 0.000,B 0.000,C 90.000,E1 40.987} C_DIS
LIN {X -0.059,Y -595.406,Z 1213.021,A 0.000,B 0.000,C 90.000,E1 39.688} C_DIS
LIN {X -0.003,Y -594.474,Z 1213.015,A 0.000,B 0.000,C 90.000,E1 38.624} C_DIS
LIN {X -0.051,Y -593.471,Z 1213.009,A 0.000,B 0.000,C 90.000,E1 37.569} C_DIS
LIN {X 0.202,Y -591.817,Z 1213.001,A 0.000,B 0.000,C 90.000,E1 36.217} C_DIS
LIN {X -0.122,Y -590.088,Z 1212.995,A 0.000,B 0.000,C 90.000,E1 35.185} C_DIS
LIN {X 0.289,Y -589.132,Z 1212.993,A 0.000,B 0.000,C 90.000,E1 34.612} C_DIS
LIN {X 0.068,Y -587.394,Z 1212.988,A 0.000,B 0.000,C 90.000,E1 33.833} C_DIS
LIN {X -0.007,Y -585.470,Z 1212.984,A 0.000,B 0.000,C 90.000,E1 33.038} C_DIS
LIN {X 0.042,Y -583.943,Z 1212.981,A 0.000,B 0.000,C 90.000,E1 32.498} C_DIS
LIN {X 0.252,Y -581.467,Z 1212.976,A 0.000,B 0.000,C 90.000,E1 31.671} C_DIS
LIN {X 0.128,Y -578.546,Z 1212.972,A 0.000,B 0.000,C 90.000,E1 30.875} C_DIS
LIN {X 0.128,Y -576.426,Z 1212.969,A 0.000,B 0.000,C 90.000,E1 30.335} C_DIS
LIN {X -0.046,Y -572.760,Z 1212.964,A 0.000,B 0.000,C 90.000,E1 29.539} C_DIS
LIN {X -0.012,Y -570.831,Z 1212.962,A 0.000,B 0.000,C 90.000,E1 29.127} C_DIS
LIN {X 0.060,Y -567.243,Z 1212.958,A 0.000,B 0.000,C 90.000,E1 28.437} C_DIS
LIN {X -0.219,Y -562.556,Z 1212.953,A 0.000,B 0.000,C 90.000,E1 27.641} C_DIS
LIN {X -0.160,Y -556.513,Z 1212.948,A 0.000,B 0.000,C 90.000,E1 26.668} C_DIS
LIN {X 0.020,Y -553.741,Z 1212.946,A 0.000,B 0.000,C 90.000,E1 26.232} C_DIS
LIN {X -0.157,Y -547.777,Z 1212.941,A 0.000,B 0.000,C 90.000,E1 25.412} C_DIS
LIN {X -0.040,Y -542.219,Z 1212.937,A 0.000,B 0.000,C 90.000,E1 24.695} C_DIS
LIN {X 0.287,Y -536.330,Z 1212.933,A 0.000,B 0.000,C 90.000,E1 23.951} C_DIS
LIN {X 0.215,Y -531.334,Z 1212.930,A 0.000,B 0.000,C 90.000,E1 23.387} C_DIS
LIN {X -0.211,Y -523.653,Z 1212.925,A 0.000,B 0.000,C 90.000,E1 22.589} C_DIS
LIN {X 0.019,Y -514.311,Z 1212.920,A 0.000,B 0.000,C 90.000,E1 21.589} C_DIS
LIN {X 0.185,Y -504.752,Z 1212.915,A 0.000,B 0.000,C 90.000,E1 20.610} C_DIS
LIN {X -0.011,Y -494.753,Z 1212.909,A 0.000,B 0.000,C 90.000,E1 19.685} C_DIS
LIN {X -0.198,Y -486.079,Z 1212.905,A 0.000,B 0.000,C 90.000,E1 18.906} C_DIS
LIN {X 0.122,Y -475.775,Z 1212.900,A 0.000,B 0.000,C 90.000,E1 17.946} C_DIS
LIN {X 0.148,Y -460.851,Z 1212.892,A 0.000,B 0.000,C 90.000,E1 16.622} C_DIS
LIN {X 0.160,Y -437.406,Z 1212.880,A 0.000,B 0.000,C 90.000,E1 14.426} C_DIS
LIN {X -0.150,Y -423.128,Z 1212.872,A 0.000,B 0.000,C 90.000,E1 13.008} C_DIS
LIN {X 0.047,Y -406.295,Z 1212.862,A 0.000,B 0.000,C 90.000,E1 11.074} C_DIS
LIN {X -0.110,Y -399.595,Z 1212.857,A 0.000,B 0.000,C 90.000,E1 10.254} C_DIS
LIN {X -0.119,Y -397.055,Z 1212.855,A 0.000,B 0.000,C 90.000,E1 9.905} C_DIS
LIN {X 0.035,Y -394.623,Z 1212.853,A 0.000,B 0.000,C 90.000,E1 9.443} C_DIS
LIN {X 0.022,Y -394.037,Z 1212.852,A 0.000,B 0.000,C 90.000,E1 9.265} C_DIS
LIN {X -0.027,Y -393.568,Z 1212.851,A 0.000,B 0.000,C 90.000,E1 9.095} C_DIS
LIN {X -0.064,Y -393.567,Z 1212.850,A 0.000,B 0.000,C 90.000,E1 9.095} C_DIS
LIN {X 0.127,Y -393.877,Z 1212.849,A 0.000,B 0.000,C 90.000,E1 8.746} C_DIS
LIN {X 0.089,Y -393.886,Z 1212.849,A 0.000,B 0.000,C 90.000,E1 8.746} C_DIS
LIN {X -0.136,Y -397.104,Z 1212.845,A 0.000,B 0.000,C 90.000,E1 8.049} C_DIS
LIN {X 0.145,Y -400.949,Z 1212.842,A 0.000,B 0.000,C 90.000,E1 7.530} C_DIS
LIN {X 0.078,Y -405.993,Z 1212.839,A 0.000,B 0.000,C 90.000,E1 7.068} C_DIS
LIN {X -0.027,Y -424.763,Z 1212.831,A 0.000,B 0.000,C 90.000,E1 5.625} C_DIS
LIN {X 0.022,Y -437.487,Z 1212.826,A 0.000,B 0.000,C 90.000,E1 4.645} C_DIS
LIN {X 0.107,Y -450.171,Z 1212.821,A 0.000,B 0.000,C 90.000,E1 3.669} C_DIS
LIN {X 0.001,Y -461.056,Z 1212.816,A 0.000,B 0.000,C 90.000,E1 2.865} C_DIS
LIN {X -0.217,Y -468.809,Z 1212.813,A 0.000,B 0.000,C 90.000,E1 2.293} C_DIS
LIN {X -0.089,Y -476.400,Z 1212.809,A 0.000,B 0.000,C 90.000,E1 1.661} C_DIS
LIN {X -0.090,Y -482.322,Z 1212.806,A 0.000,B 0.000,C 90.000,E1 1.146} C_DIS
LIN {X 0.227,Y -486.300,Z 1212.804,A 0.000,B 0.000,C 90.000,E1 0.745} C_DIS
LIN {X 0.050,Y -491.898,Z 1212.801,A 0.000,B 0.000,C 90.000,E1 0.229} C_DIS
LIN {X 0.216,Y -498.804,Z 1212.797,A 0.000,B 0.000,C 90.000,E1 359.484} C_DIS
LIN {X -0.145,Y -505.183,Z 1212.793,A 0.000,B 0.000,C 90.000,E1 358.797} C_DIS
LIN {X -0.013,Y -511.077,Z 1212.789,A 0.000,B 0.000,C 90.000,E1 358.051} C_DIS
LIN {X 0.146,Y -516.509,Z 1212.785,A 0.000,B 0.000,C 90.000,E1 357.306} C_DIS
LIN {X 0.036,Y -520.653,Z 1212.782,A 0.000,B 0.000,C 90.000,E1 356.731} C_DIS
LIN {X 0.162,Y -525.388,Z 1212.778,A 0.000,B 0.000,C 90.000,E1 355.988} C_DIS
LIN {X 0.119,Y -528.900,Z 1212.775,A 0.000,B 0.000,C 90.000,E1 355.412} C_DIS
LIN {X -0.174,Y -532.854,Z 1212.771,A 0.000,B 0.000,C 90.000,E1 354.723} C_DIS
LIN {X 0.152,Y -536.442,Z 1212.767,A 0.000,B 0.000,C 90.000,E1 353.970} C_DIS
LIN {X -0.075,Y -539.696,Z 1212.763,A 0.000,B 0.000,C 90.000,E1 353.280} C_DIS
LIN {X -0.282,Y -542.641,Z 1212.759,A 0.000,B 0.000,C 90.000,E1 352.591} C_DIS
LIN {X -0.132,Y -544.872,Z 1212.756,A 0.000,B 0.000,C 90.000,E1 352.008} C_DIS
LIN {X 0.054,Y -547.864,Z 1212.751,A 0.000,B 0.000,C 90.000,E1 351.141} C_DIS
LIN {X -0.275,Y -550.548,Z 1212.746,A 0.000,B 0.000,C 90.000,E1 350.330} C_DIS
LIN {X 0.180,Y -553.813,Z 1212.740,A 0.000,B 0.000,C 90.000,E1 349.162} C_DIS
LIN {X 0.146,Y -556.757,Z 1212.734,A 0.000,B 0.000,C 90.000,E1 348.049} C_DIS
LIN {X 0.012,Y -558.866,Z 1212.729,A 0.000,B 0.000,C 90.000,E1 347.229} C_DIS
LIN {X 0.190,Y -561.948,Z 1212.721,A 0.000,B 0.000,C 90.000,E1 345.825} C_DIS
LIN {X 0.155,Y -564.755,Z 1212.714,A 0.000,B 0.000,C 90.000,E1 344.448} C_DIS
LIN {X -0.141,Y -566.861,Z 1212.708,A 0.000,B 0.000,C 90.000,E1 343.378} C_DIS
LIN {X 0.299,Y -568.720,Z 1212.702,A 0.000,B 0.000,C 90.000,E1 342.236} C_DIS
LIN {X -0.120,Y -570.009,Z 1212.697,A 0.000,B 0.000,C 90.000,E1 341.456} C_DIS
LIN {X 0.196,Y -571.132,Z 1212.692,A 0.000,B 0.000,C 90.000,E1 340.604} C_DIS
LIN {X 0.148,Y -572.419,Z 1212.686,A 0.000,B 0.000,C 90.000,E1 339.518} C_DIS
LIN {X -0.220,Y -573.384,Z 1212.680,A 0.000,B 0.000,C 90.000,E1 338.465} C_DIS
LIN {X 0.124,Y -573.742,Z 1212.676,A 0.000,B 0.000,C 90.000,E1 337.614} C_DIS
LIN {X 0.160,Y -573.840,Z 1212.671,A 0.000,B 0.000,C 90.000,E1 336.794} C_DIS
LIN {X -0.162,Y -573.774,Z 1212.668,A 0.000,B 0.000,C 90.000,E1 336.282} C_DIS
LIN {X 0.006,Y -573.122,Z 1212.662,A 0.000,B 0.000,C 90.000,E1 335.177} C_DIS
LIN {X -0.317,Y -572.648,Z 1212.659,A 0.000,B 0.000,C 90.000,E1 334.665} C_DIS
LIN {X -0.038,Y -571.447,Z 1212.655,A 0.000,B 0.000,C 90.000,E1 333.819} C_DIS
LIN {X 0.144,Y -570.451,Z 1212.652,A 0.000,B 0.000,C 90.000,E1 333.256} C_DIS
LIN {X 0.142,Y -568.601,Z 1212.647,A 0.000,B 0.000,C 90.000,E1 332.436} C_DIS
LIN {X -0.121,Y -566.543,Z 1212.642,A 0.000,B 0.000,C 90.000,E1 331.641} C_DIS
LIN {X 0.096,Y -564.015,Z 1212.638,A 0.000,B 0.000,C 90.000,E1 330.795} C_DIS
LIN {X -0.305,Y -560.032,Z 1212.632,A 0.000,B 0.000,C 90.000,E1 329.871} C_DIS
LIN {X 0.222,Y -556.479,Z 1212.629,A 0.000,B 0.000,C 90.000,E1 329.125} C_DIS
LIN {X -0.047,Y -552.397,Z 1212.625,A 0.000,B 0.000,C 90.000,E1 328.456} C_DIS
LIN {X 0.239,Y -548.723,Z 1212.622,A 0.000,B 0.000,C 90.000,E1 327.867} C_DIS
LIN {X 0.062,Y -542.650,Z 1212.617,A 0.000,B 0.000,C 90.000,E1 327.041} C_DIS
LIN {X -0.047,Y -539.437,Z 1212.615,A 0.000,B 0.000,C 90.000,E1 326.628} C_DIS
LIN {X -0.165,Y -533.662,Z 1212.611,A 0.000,B 0.000,C 90.000,E1 325.928} C_DIS
LIN {X -0.159,Y -519.536,Z 1212.601,A 0.000,B 0.000,C 90.000,E1 324.196} C_DIS
LIN {X -0.083,Y -516.357,Z 1212.599,A 0.000,B 0.000,C 90.000,E1 323.749} C_DIS
LIN {X 0.083,Y -513.728,Z 1212.596,A 0.000,B 0.000,C 90.000,E1 323.290} C_DIS
LIN {X -0.143,Y -510.948,Z 1212.593,A 0.000,B 0.000,C 90.000,E1 322.683} C_DIS
LIN {X 0.092,Y -509.755,Z 1212.589,A 0.000,B 0.000,C 90.000,E1 322.065} C_DIS
LIN {X 0.004,Y -509.379,Z 1212.588,A 0.000,B 0.000,C 90.000,E1 321.778} C_DIS
LIN {X 0.045,Y -509.094,Z 1212.583,A 0.000,B 0.000,C 90.000,E1 320.884} C_DIS
LIN {X 0.129,Y -509.735,Z 1212.573,A 0.000,B 0.000,C 90.000,E1 319.094} C_DIS
LIN {X 0.035,Y -510.499,Z 1212.566,A 0.000,B 0.000,C 90.000,E1 317.919} C_DIS
LIN {X 0.005,Y -511.696,Z 1212.555,A 0.000,B 0.000,C 90.000,E1 315.850} C_DIS
LIN {X -0.067,Y -512.375,Z 1212.548,A 0.000,B 0.000,C 90.000,E1 314.676} C_DIS
LIN {X -0.069,Y -513.418,Z 1212.537,A 0.000,B 0.000,C 90.000,E1 312.609} C_DIS
LIN {X -0.192,Y -514.176,Z 1212.529,A 0.000,B 0.000,C 90.000,E1 311.148} C_DIS
LIN {X 0.014,Y -515.093,Z 1212.519,A 0.000,B 0.000,C 90.000,E1 309.358} C_DIS
LIN {X -0.014,Y -515.697,Z 1212.510,A 0.000,B 0.000,C 90.000,E1 307.890} C_DIS
LIN {X 0.241,Y -516.448,Z 1212.499,A 0.000,B 0.000,C 90.000,E1 305.804} C_DIS
LIN {X 0.042,Y -517.150,Z 1212.491,A 0.000,B 0.000,C 90.000,E1 304.358} C_DIS
LIN {X 0.143,Y -517.700,Z 1212.483,A 0.000,B 0.000,C 90.000,E1 302.880} C_DIS
LIN {X 0.124,Y -518.187,Z 1212.475,A 0.000,B 0.000,C 90.000,E1 301.416} C_DIS
LIN {X 0.013,Y -518.434,Z 1212.468,A 0.000,B 0.000,C 90.000,E1 300.256} C_DIS
LIN {X 0.122,Y -518.680,Z 1212.458,A 0.000,B 0.000,C 90.000,E1 298.487} C_DIS
LIN {X -0.043,Y -518.804,Z 1212.452,A 0.000,B 0.000,C 90.000,E1 297.334} C_DIS
LIN {X 0.028,Y -518.912,Z 1212.445,A 0.000,B 0.000,C 90.000,E1 296.155} C_DIS
LIN {X 0.136,Y -518.951,Z 1212.436,A 0.000,B 0.000,C 90.000,E1 294.387} C_DIS
LIN {X 0.036,Y -519.007,Z 1212.426,A 0.000,B 0.000,C 90.000,E1 292.642} C_DIS
LIN {X -0.015,Y -519.080,Z 1212.421,A 0.000,B 0.000,C 90.000,E1 291.770} C_DIS
LIN {X -0.257,Y -518.938,Z 1212.416,A 0.000,B 0.000,C 90.000,E1 290.918} C_DIS
LIN {X -0.073,Y -518.374,Z 1212.406,A 0.000,B 0.000,C 90.000,E1 289.141} C_DIS
LIN {X -0.217,Y -517.600,Z 1212.398,A 0.000,B 0.000,C 90.000,E1 287.692} C_DIS
LIN {X -0.031,Y -516.817,Z 1212.390,A 0.000,B 0.000,C 90.000,E1 286.205} C_DIS
LIN {X 0.235,Y -515.527,Z 1212.379,A 0.000,B 0.000,C 90.000,E1 284.120} C_DIS
LIN {X 0.252,Y -514.620,Z 1212.370,A 0.000,B 0.000,C 90.000,E1 282.647} C_DIS
LIN {X 0.141,Y -513.615,Z 1212.362,A 0.000,B 0.000,C 90.000,E1 281.186} C_DIS
LIN {X -0.130,Y -512.404,Z 1212.351,A 0.000,B 0.000,C 90.000,E1 279.151} C_DIS
LIN {X -0.041,Y -510.932,Z 1212.338,A 0.000,B 0.000,C 90.000,E1 276.777} C_DIS
LIN {X 0.032,Y -509.912,Z 1212.328,A 0.000,B 0.000,C 90.000,E1 274.992} C_DIS
LIN {X 0.138,Y -509.001,Z 1212.320,A 0.000,B 0.000,C 90.000,E1 273.498} C_DIS
LIN {X -0.074,Y -507.637,Z 1212.306,A 0.000,B 0.000,C 90.000,E1 271.146} C_DIS
LIN {X -0.152,Y -506.626,Z 1212.297,A 0.000,B 0.000,C 90.000,E1 269.370} C_DIS
LIN {X -0.035,Y -505.940,Z 1212.290,A 0.000,B 0.000,C 90.000,E1 268.165} C_DIS
LIN {X -0.029,Y -505.027,Z 1212.281,A 0.000,B 0.000,C 90.000,E1 266.674} C_DIS
LIN {X -0.011,Y -504.047,Z 1212.273,A 0.000,B 0.000,C 90.000,E1 265.179} C_DIS
LIN {X -0.088,Y -502.627,Z 1212.263,A 0.000,B 0.000,C 90.000,E1 263.394} C_DIS
LIN {X 0.055,Y -500.149,Z 1212.248,A 0.000,B 0.000,C 90.000,E1 260.679} C_DIS
LIN {X 0.021,Y -498.418,Z 1212.237,A 0.000,B 0.000,C 90.000,E1 258.578} C_DIS
LIN {X -0.038,Y -496.551,Z 1212.223,A 0.000,B 0.000,C 90.000,E1 256.172} C_DIS
LIN {X 0.044,Y -495.058,Z 1212.211,A 0.000,B 0.000,C 90.000,E1 254.047} C_DIS
LIN {X 0.018,Y -494.375,Z 1212.206,A 0.000,B 0.000,C 90.000,E1 253.142} C_DIS
LIN {X -0.037,Y -493.504,Z 1212.196,A 0.000,B 0.000,C 90.000,E1 251.329} C_DIS
LIN {X -0.030,Y -492.874,Z 1212.190,A 0.000,B 0.000,C 90.000,E1 250.115} C_DIS
LIN {X 0.003,Y -491.891,Z 1212.181,A 0.000,B 0.000,C 90.000,E1 248.592} C_DIS
LIN {X 0.188,Y -490.769,Z 1212.173,A 0.000,B 0.000,C 90.000,E1 247.050} C_DIS
LIN {X 0.093,Y -489.304,Z 1212.164,A 0.000,B 0.000,C 90.000,E1 245.537} C_DIS
LIN {X -0.046,Y -488.029,Z 1212.157,A 0.000,B 0.000,C 90.000,E1 244.332} C_DIS
LIN {X 0.025,Y -486.407,Z 1212.149,A 0.000,B 0.000,C 90.000,E1 242.794} C_DIS
LIN {X 0.069,Y -483.506,Z 1212.135,A 0.000,B 0.000,C 90.000,E1 240.333} C_DIS
LIN {X 0.093,Y -481.602,Z 1212.127,A 0.000,B 0.000,C 90.000,E1 238.791} C_DIS
LIN {X -0.113,Y -479.329,Z 1212.116,A 0.000,B 0.000,C 90.000,E1 236.962} C_DIS
LIN {X 0.089,Y -477.540,Z 1212.108,A 0.000,B 0.000,C 90.000,E1 235.388} C_DIS
LIN {X 0.106,Y -475.076,Z 1212.096,A 0.000,B 0.000,C 90.000,E1 233.210} C_DIS
LIN {X 0.169,Y -473.017,Z 1212.085,A 0.000,B 0.000,C 90.000,E1 231.331} C_DIS
LIN {X 0.035,Y -471.416,Z 1212.077,A 0.000,B 0.000,C 90.000,E1 229.784} C_DIS
LIN {X -0.099,Y -469.557,Z 1212.066,A 0.000,B 0.000,C 90.000,E1 227.919} C_DIS
LIN {X -0.022,Y -467.971,Z 1212.057,A 0.000,B 0.000,C 90.000,E1 226.338} C_DIS
LIN {X 0.164,Y -466.051,Z 1212.045,A 0.000,B 0.000,C 90.000,E1 224.109} C_DIS
LIN {X 0.036,Y -464.528,Z 1212.031,A 0.000,B 0.000,C 90.000,E1 221.595} C_DIS
LIN {X -0.004,Y -464.690,Z 1212.001,A 0.000,B 0.000,C 90.000,E1 216.217} C_DIS
LIN {X -0.124,Y -466.173,Z 1211.982,A 0.000,B 0.000,C 90.000,E1 212.752} C_DIS
LIN {X -0.102,Y -468.161,Z 1211.970,A 0.000,B 0.000,C 90.000,E1 210.541} C_DIS
LIN {X 0.004,Y -471.570,Z 1211.952,A 0.000,B 0.000,C 90.000,E1 207.385} C_DIS
LIN {X 0.073,Y -472.676,Z 1211.947,A 0.000,B 0.000,C 90.000,E1 206.437} C_DIS
LIN {X -0.100,Y -474.263,Z 1211.940,A 0.000,B 0.000,C 90.000,E1 205.207} C_DIS
LIN {X -0.099,Y -477.261,Z 1211.928,A 0.000,B 0.000,C 90.000,E1 203.025} C_DIS
LIN {X 0.109,Y -485.258,Z 1211.904,A 0.000,B 0.000,C 90.000,E1 198.671} C_DIS
LIN {X -0.107,Y -490.208,Z 1211.892,A 0.000,B 0.000,C 90.000,E1 196.551} C_DIS
LIN {X -0.040,Y -494.898,Z 1211.882,A 0.000,B 0.000,C 90.000,E1 194.717} C_DIS
LIN {X 0.141,Y -499.925,Z 1211.872,A 0.000,B 0.000,C 90.000,E1 192.883} C_DIS
LIN {X -0.215,Y -504.312,Z 1211.863,A 0.000,B 0.000,C 90.000,E1 191.422} C_DIS
LIN {X 0.009,Y -508.623,Z 1211.855,A 0.000,B 0.000,C 90.000,E1 189.905} C_DIS
LIN {X 0.166,Y -515.070,Z 1211.844,A 0.000,B 0.000,C 90.000,E1 187.814} C_DIS
LIN {X -0.060,Y -518.785,Z 1211.837,A 0.000,B 0.000,C 90.000,E1 186.663} C_DIS
LIN {X -0.228,Y -522.394,Z 1211.831,A 0.000,B 0.000,C 90.000,E1 185.511} C_DIS
LIN {X 0.103,Y -528.593,Z 1211.819,A 0.000,B 0.000,C 90.000,E1 183.440} C_DIS
LIN {X 0.024,Y -533.017,Z 1211.811,A 0.000,B 0.000,C 90.000,E1 182.007} C_DIS
LIN {X 0.023,Y -537.472,Z 1211.803,A 0.000,B 0.000,C 90.000,E1 180.573} C_DIS
LIN {X 0.070,Y -541.022,Z 1211.797,A 0.000,B 0.000,C 90.000,E1 179.427} C_DIS
LIN {X 0.214,Y -545.333,Z 1211.789,A 0.000,B 0.000,C 90.000,E1 177.993} C_DIS
LIN {X -0.060,Y -550.369,Z 1211.780,A 0.000,B 0.000,C 90.000,E1 176.331} C_DIS
LIN {X -0.264,Y -554.360,Z 1211.772,A 0.000,B 0.000,C 90.000,E1 174.951} C_DIS
LIN {X 0.150,Y -558.317,Z 1211.764,A 0.000,B 0.000,C 90.000,E1 173.514} C_DIS
LIN {X -0.116,Y -563.652,Z 1211.753,A 0.000,B 0.000,C 90.000,E1 171.602} C_DIS
LIN {X 0.135,Y -568.218,Z 1211.744,A 0.000,B 0.000,C 90.000,E1 169.926} C_DIS
LIN {X -0.244,Y -573.450,Z 1211.734,A 0.000,B 0.000,C 90.000,E1 168.049} C_DIS
LIN {X 0.069,Y -578.770,Z 1211.723,A 0.000,B 0.000,C 90.000,E1 166.117} C_DIS
LIN {X 0.235,Y -584.278,Z 1211.713,A 0.000,B 0.000,C 90.000,E1 164.212} C_DIS
LIN {X 0.297,Y -589.114,Z 1211.703,A 0.000,B 0.000,C 90.000,E1 162.598} C_DIS
LIN {X 0.060,Y -598.481,Z 1211.687,A 0.000,B 0.000,C 90.000,E1 159.699} C_DIS
LIN {X 0.166,Y -604.989,Z 1211.677,A 0.000,B 0.000,C 90.000,E1 157.847} C_DIS
LIN {X 0.252,Y -608.709,Z 1211.671,A 0.000,B 0.000,C 90.000,E1 156.794} C_DIS
LIN {X -0.210,Y -613.286,Z 1211.664,A 0.000,B 0.000,C 90.000,E1 155.537} C_DIS
LIN {X -0.049,Y -617.649,Z 1211.657,A 0.000,B 0.000,C 90.000,E1 154.229} C_DIS
LIN {X -0.104,Y -621.050,Z 1211.651,A 0.000,B 0.000,C 90.000,E1 153.204} C_DIS
LIN {X 0.177,Y -624.306,Z 1211.645,A 0.000,B 0.000,C 90.000,E1 152.153} C_DIS
LIN {X 0.020,Y -629.831,Z 1211.635,A 0.000,B 0.000,C 90.000,E1 150.383} C_DIS
LIN {X -0.050,Y -634.404,Z 1211.627,A 0.000,B 0.000,C 90.000,E1 148.869} C_DIS
LIN {X -0.128,Y -637.295,Z 1211.621,A 0.000,B 0.000,C 90.000,E1 147.867} C_DIS
LIN {X 0.176,Y -640.152,Z 1211.616,A 0.000,B 0.000,C 90.000,E1 146.834} C_DIS
LIN {X -0.370,Y -642.741,Z 1211.610,A 0.000,B 0.000,C 90.000,E1 145.881} C_DIS
LIN {X -0.105,Y -645.853,Z 1211.603,A 0.000,B 0.000,C 90.000,E1 144.609} C_DIS
LIN {X 0.218,Y -648.630,Z 1211.596,A 0.000,B 0.000,C 90.000,E1 143.336} C_DIS
LIN {X 0.066,Y -651.284,Z 1211.590,A 0.000,B 0.000,C 90.000,E1 142.110} C_DIS
LIN {X -0.048,Y -653.945,Z 1211.583,A 0.000,B 0.000,C 90.000,E1 140.884} C_DIS
LIN {X 0.205,Y -657.551,Z 1211.573,A 0.000,B 0.000,C 90.000,E1 139.138} C_DIS
LIN {X 0.084,Y -660.751,Z 1211.565,A 0.000,B 0.000,C 90.000,E1 137.676} C_DIS
LIN {X 0.006,Y -664.411,Z 1211.555,A 0.000,B 0.000,C 90.000,E1 135.972} C_DIS
LIN {X -0.008,Y -668.870,Z 1211.545,A 0.000,B 0.000,C 90.000,E1 134.028} C_DIS
LIN {X 0.121,Y -673.684,Z 1211.534,A 0.000,B 0.000,C 90.000,E1 132.081} C_DIS
LIN {X -0.103,Y -677.809,Z 1211.525,A 0.000,B 0.000,C 90.000,E1 130.415} C_DIS
LIN {X 0.126,Y -680.785,Z 1211.518,A 0.000,B 0.000,C 90.000,E1 129.197} C_DIS
LIN {X -0.037,Y -683.751,Z 1211.511,A 0.000,B 0.000,C 90.000,E1 128.016} C_DIS
LIN {X 0.224,Y -688.559,Z 1211.501,A 0.000,B 0.000,C 90.000,E1 126.091} C_DIS
LIN {X -0.039,Y -691.850,Z 1211.493,A 0.000,B 0.000,C 90.000,E1 124.692} C_DIS
LIN {X 0.461,Y -694.003,Z 1211.488,A 0.000,B 0.000,C 90.000,E1 123.706} C_DIS
LIN {X 0.253,Y -696.635,Z 1211.481,A 0.000,B 0.000,C 90.000,E1 122.546} C_DIS
LIN {X 0.058,Y -698.583,Z 1211.476,A 0.000,B 0.000,C 90.000,E1 121.623} C_DIS
LIN {X -0.082,Y -700.849,Z 1211.469,A 0.000,B 0.000,C 90.000,E1 120.463} C_DIS
LIN {X 0.058,Y -703.038,Z 1211.463,A 0.000,B 0.000,C 90.000,E1 119.283} C_DIS
LIN {X -0.052,Y -704.564,Z 1211.458,A 0.000,B 0.000,C 90.000,E1 118.359} C_DIS
LIN {X -0.102,Y -705.219,Z 1211.455,A 0.000,B 0.000,C 90.000,E1 117.897} C_DIS
LIN {X -0.152,Y -705.746,Z 1211.452,A 0.000,B 0.000,C 90.000,E1 117.436} C_DIS
LIN {X 0.064,Y -706.365,Z 1211.447,A 0.000,B 0.000,C 90.000,E1 116.488} C_DIS
LIN {X 0.002,Y -706.708,Z 1211.443,A 0.000,B 0.000,C 90.000,E1 115.796} C_DIS
LIN {X 0.248,Y -706.669,Z 1211.439,A 0.000,B 0.000,C 90.000,E1 115.079} C_DIS
LIN {X -0.104,Y -706.334,Z 1211.437,A 0.000,B 0.000,C 90.000,E1 114.643} C_DIS
LIN {X 0.189,Y -705.586,Z 1211.434,A 0.000,B 0.000,C 90.000,E1 114.155} C_DIS
LIN {X -0.165,Y -705.135,Z 1211.433,A 0.000,B 0.000,C 90.000,E1 113.951} C_DIS
LIN {X 0.125,Y -703.034,Z 1211.430,A 0.000,B 0.000,C 90.000,E1 113.462} C_DIS
LIN {X 0.265,Y -702.486,Z 1211.430,A 0.000,B 0.000,C 90.000,E1 113.334} C_DIS
LIN {X -0.239,Y -701.776,Z 1211.429,A 0.000,B 0.000,C 90.000,E1 113.259} C_DIS
LIN {X -0.103,Y -700.715,Z 1211.428,A 0.000,B 0.000,C 90.000,E1 113.131} C_DIS
LIN {X -0.048,Y -695.246,Z 1211.426,A 0.000,B 0.000,C 90.000,E1 112.695} C_DIS
LIN {X -0.012,Y -693.537,Z 1211.426,A 0.000,B 0.000,C 90.000,E1 112.589} C_DIS
LIN {X 0.261,Y -686.677,Z 1211.424,A 0.000,B 0.000,C 90.000,E1 112.333} C_DIS
LIN {X -0.220,Y -684.732,Z 1211.424,A 0.000,B 0.000,C 90.000,E1 112.333} C_DIS
LIN {X 0.052,Y -676.932,Z 1211.424,A 0.000,B 0.000,C 90.000,E1 112.280} C_DIS
LIN {X 0.003,Y -610.647,Z 1211.424,A 0.000,B 0.000,C 90.000,E1 112.280} C_DIS
LIN {X -0.116,Y -608.960,Z 1211.423,A 0.000,B 0.000,C 90.000,E1 112.206} C_DIS
LIN {X -0.254,Y -603.548,Z 1211.421,A 0.000,B 0.000,C 90.000,E1 111.844} C_DIS
LIN {X 0.145,Y -599.708,Z 1211.419,A 0.000,B 0.000,C 90.000,E1 111.482} C_DIS
LIN {X -0.153,Y -596.144,Z 1211.417,A 0.000,B 0.000,C 90.000,E1 111.153} C_DIS
LIN {X 0.136,Y -594.441,Z 1211.416,A 0.000,B 0.000,C 90.000,E1 110.865} C_DIS
LIN {X -0.124,Y -594.086,Z 1211.416,A 0.000,B 0.000,C 90.000,E1 110.844} C_DIS
LIN {X -0.167,Y -594.074,Z 1211.416,A 0.000,B 0.000,C 90.000,E1 110.844} C_DIS
LIN {X 0.033,Y -593.934,Z 1211.415,A 0.000,B 0.000,C 90.000,E1 110.610} C_DIS
LIN {X -0.336,Y -594.736,Z 1211.412,A 0.000,B 0.000,C 90.000,E1 110.248} C_DIS
LIN {X 0.245,Y -598.366,Z 1211.406,A 0.000,B 0.000,C 90.000,E1 109.141} C_DIS
LIN {X -0.171,Y -601.277,Z 1211.401,A 0.000,B 0.000,C 90.000,E1 108.127} C_DIS
LIN {X 0.216,Y -604.282,Z 1211.395,A 0.000,B 0.000,C 90.000,E1 107.040} C_DIS
LIN {X 0.153,Y -606.363,Z 1211.391,A 0.000,B 0.000,C 90.000,E1 106.260} C_DIS
LIN {X 0.207,Y -607.638,Z 1211.388,A 0.000,B 0.000,C 90.000,E1 105.733} C_DIS
LIN {X -0.152,Y -608.734,Z 1211.385,A 0.000,B 0.000,C 90.000,E1 105.245} C_DIS
LIN {X -0.334,Y -609.907,Z 1211.380,A 0.000,B 0.000,C 90.000,E1 104.481} C_DIS
LIN {X -0.100,Y -610.492,Z 1211.377,A 0.000,B 0.000,C 90.000,E1 103.939} C_DIS
LIN {X -0.011,Y -610.814,Z 1211.375,A 0.000,B 0.000,C 90.000,E1 103.411} C_DIS
LIN {X -0.262,Y -610.821,Z 1211.373,A 0.000,B 0.000,C 90.000,E1 103.175} C_DIS
LIN {X -0.169,Y -610.574,Z 1211.370,A 0.000,B 0.000,C 90.000,E1 102.647} C_DIS
LIN {X -0.077,Y -610.051,Z 1211.367,A 0.000,B 0.000,C 90.000,E1 102.119} C_DIS
LIN {X 0.011,Y -608.949,Z 1211.365,A 0.000,B 0.000,C 90.000,E1 101.591} C_DIS
LIN {X -0.025,Y -607.555,Z 1211.362,A 0.000,B 0.000,C 90.000,E1 101.074} C_DIS
LIN {X -0.285,Y -606.751,Z 1211.360,A 0.000,B 0.000,C 90.000,E1 100.838} C_DIS
LIN {X -0.218,Y -604.657,Z 1211.357,A 0.000,B 0.000,C 90.000,E1 100.310} C_DIS
LIN {X -0.170,Y -602.087,Z 1211.354,A 0.000,B 0.000,C 90.000,E1 99.782} C_DIS
LIN {X 0.154,Y -597.948,Z 1211.351,A 0.000,B 0.000,C 90.000,E1 99.095} C_DIS
LIN {X 0.147,Y -594.118,Z 1211.348,A 0.000,B 0.000,C 90.000,E1 98.568} C_DIS
LIN {X 0.026,Y -589.834,Z 1211.345,A 0.000,B 0.000,C 90.000,E1 98.049} C_DIS
LIN {X 0.116,Y -586.089,Z 1211.343,A 0.000,B 0.000,C 90.000,E1 97.644} C_DIS
LIN {X -0.178,Y -583.209,Z 1211.341,A 0.000,B 0.000,C 90.000,E1 97.409} C_DIS
LIN {X 0.227,Y -578.919,Z 1211.339,A 0.000,B 0.000,C 90.000,E1 97.011} C_DIS
LIN {X -0.281,Y -575.635,Z 1211.338,A 0.000,B 0.000,C 90.000,E1 96.834} C_DIS
LIN {X 0.097,Y -571.112,Z 1211.336,A 0.000,B 0.000,C 90.000,E1 96.486} C_DIS
LIN {X -0.144,Y -568.434,Z 1211.335,A 0.000,B 0.000,C 90.000,E1 96.315} C_DIS
LIN {X -0.194,Y -565.063,Z 1211.333,A 0.000,B 0.000,C 90.000,E1 95.967} C_DIS
LIN {X -0.178,Y -563.597,Z 1211.332,A 0.000,B 0.000,C 90.000,E1 95.796} C_DIS
LIN {X -0.215,Y -563.583,Z 1211.332,A 0.000,B 0.000,C 90.000,E1 95.796} C_DIS
LIN {X 0.021,Y -563.339,Z 1211.331,A 0.000,B 0.000,C 90.000,E1 95.568} C_DIS
LIN {X 0.263,Y -563.332,Z 1211.330,A 0.000,B 0.000,C 90.000,E1 95.391} C_DIS
LIN {X -0.205,Y -563.132,Z 1211.329,A 0.000,B 0.000,C 90.000,E1 95.163} C_DIS
LIN {X -0.229,Y -563.270,Z 1211.323,A 0.000,B 0.000,C 90.000,E1 94.069} C_DIS
LIN {X -0.154,Y -564.269,Z 1211.313,A 0.000,B 0.000,C 90.000,E1 92.407} C_DIS
LIN {X -0.270,Y -565.081,Z 1211.307,A 0.000,B 0.000,C 90.000,E1 91.318} C_DIS
LIN {X -0.274,Y -566.073,Z 1211.300,A 0.000,B 0.000,C 90.000,E1 89.943} C_DIS
LIN {X 0.111,Y -567.728,Z 1211.287,A 0.000,B 0.000,C 90.000,E1 87.707} C_DIS
LIN {X -0.123,Y -569.143,Z 1211.277,A 0.000,B 0.000,C 90.000,E1 85.812} C_DIS
LIN {X 0.292,Y -570.703,Z 1211.266,A 0.000,B 0.000,C 90.000,E1 83.856} C_DIS
LIN {X -0.065,Y -571.812,Z 1211.259,A 0.000,B 0.000,C 90.000,E1 82.527} C_DIS
LIN {X 0.162,Y -572.890,Z 1211.251,A 0.000,B 0.000,C 90.000,E1 81.141} C_DIS
LIN {X 0.127,Y -573.999,Z 1211.242,A 0.000,B 0.000,C 90.000,E1 79.511} C_DIS
LIN {X 0.108,Y -575.051,Z 1211.233,A 0.000,B 0.000,C 90.000,E1 77.881} C_DIS
LIN {X -0.208,Y -575.922,Z 1211.224,A 0.000,B 0.000,C 90.000,E1 76.284} C_DIS
LIN {X 0.062,Y -576.756,Z 1211.215,A 0.000,B 0.000,C 90.000,E1 74.629} C_DIS
LIN {X -0.054,Y -577.620,Z 1211.206,A 0.000,B 0.000,C 90.000,E1 73.015} C_DIS
LIN {X -0.160,Y -578.555,Z 1211.197,A 0.000,B 0.000,C 90.000,E1 71.402} C_DIS
LIN {X 0.151,Y -579.941,Z 1211.185,A 0.000,B 0.000,C 90.000,E1 69.209} C_DIS
LIN {X 0.031,Y -581.879,Z 1211.171,A 0.000,B 0.000,C 90.000,E1 66.794} C_DIS
LIN {X 0.055,Y -583.397,Z 1211.162,A 0.000,B 0.000,C 90.000,E1 65.177} C_DIS
LIN {X -0.045,Y -585.126,Z 1211.152,A 0.000,B 0.000,C 90.000,E1 63.307} C_DIS
LIN {X -0.088,Y -587.030,Z 1211.141,A 0.000,B 0.000,C 90.000,E1 61.435} C_DIS
LIN {X 0.304,Y -588.652,Z 1211.132,A 0.000,B 0.000,C 90.000,E1 59.793} C_DIS
LIN {X 0.140,Y -589.679,Z 1211.126,A 0.000,B 0.000,C 90.000,E1 58.742} C_DIS
LIN {X -0.326,Y -590.871,Z 1211.119,A 0.000,B 0.000,C 90.000,E1 57.454} C_DIS
LIN {X 0.255,Y -592.119,Z 1211.110,A 0.000,B 0.000,C 90.000,E1 55.801} C_DIS
LIN {X 0.374,Y -593.383,Z 1211.101,A 0.000,B 0.000,C 90.000,E1 54.196} C_DIS
LIN {X 0.031,Y -594.559,Z 1211.093,A 0.000,B 0.000,C 90.000,E1 52.637} C_DIS
LIN {X 0.230,Y -595.144,Z 1211.088,A 0.000,B 0.000,C 90.000,E1 51.823} C_DIS
LIN {X -0.184,Y -596.175,Z 1211.079,A 0.000,B 0.000,C 90.000,E1 50.275} C_DIS
LIN {X 0.030,Y -596.771,Z 1211.072,A 0.000,B 0.000,C 90.000,E1 48.933} C_DIS
LIN {X 0.017,Y -597.316,Z 1211.063,A 0.000,B 0.000,C 90.000,E1 47.349} C_DIS
LIN {X 0.198,Y -597.523,Z 1211.059,A 0.000,B 0.000,C 90.000,E1 46.539} C_DIS
LIN {X -0.047,Y -597.723,Z 1211.051,A 0.000,B 0.000,C 90.000,E1 45.243} C_DIS
LIN {X -0.288,Y -597.504,Z 1211.044,A 0.000,B 0.000,C 90.000,E1 43.947} C_DIS
LIN {X 0.115,Y -597.120,Z 1211.038,A 0.000,B 0.000,C 90.000,E1 42.852} C_DIS
LIN {X 0.060,Y -596.246,Z 1211.029,A 0.000,B 0.000,C 90.000,E1 41.272} C_DIS
LIN {X 0.263,Y -595.343,Z 1211.022,A 0.000,B 0.000,C 90.000,E1 39.930} C_DIS
LIN {X -0.143,Y -594.505,Z 1211.016,A 0.000,B 0.000,C 90.000,E1 38.910} C_DIS
LIN {X 0.028,Y -593.169,Z 1211.009,A 0.000,B 0.000,C 90.000,E1 37.569} C_DIS
LIN {X -0.152,Y -592.232,Z 1211.004,A 0.000,B 0.000,C 90.000,E1 36.790} C_DIS
LIN {X -0.127,Y -590.719,Z 1210.998,A 0.000,B 0.000,C 90.000,E1 35.724} C_DIS
LIN {X -0.127,Y -588.817,Z 1210.993,A 0.000,B 0.000,C 90.000,E1 34.659} C_DIS
LIN {X 0.131,Y -587.074,Z 1210.988,A 0.000,B 0.000,C 90.000,E1 33.833} C_DIS
LIN {X 0.053,Y -585.137,Z 1210.984,A 0.000,B 0.000,C 90.000,E1 33.038} C_DIS
LIN {X 0.101,Y -583.610,Z 1210.981,A 0.000,B 0.000,C 90.000,E1 32.498} C_DIS
LIN {X 0.307,Y -581.082,Z 1210.976,A 0.000,B 0.000,C 90.000,E1 31.671} C_DIS
LIN {X 0.324,Y -579.195,Z 1210.973,A 0.000,B 0.000,C 90.000,E1 31.131} C_DIS
LIN {X 0.176,Y -576.003,Z 1210.969,A 0.000,B 0.000,C 90.000,E1 30.335} C_DIS
LIN {X 0.076,Y -572.955,Z 1210.965,A 0.000,B 0.000,C 90.000,E1 29.667} C_DIS
LIN {X 0.028,Y -570.371,Z 1210.962,A 0.000,B 0.000,C 90.000,E1 29.127} C_DIS
LIN {X 0.096,Y -566.772,Z 1210.958,A 0.000,B 0.000,C 90.000,E1 28.437} C_DIS
LIN {X -0.188,Y -562.055,Z 1210.953,A 0.000,B 0.000,C 90.000,E1 27.641} C_DIS
LIN {X -0.031,Y -556.905,Z 1210.949,A 0.000,B 0.000,C 90.000,E1 26.796} C_DIS
LIN {X 0.149,Y -554.222,Z 1210.947,A 0.000,B 0.000,C 90.000,E1 26.360} C_DIS
LIN {X -0.025,Y -548.272,Z 1210.942,A 0.000,B 0.000,C 90.000,E1 25.540} C_DIS
LIN {X 0.099,Y -542.816,Z 1210.938,A 0.000,B 0.000,C 90.000,E1 24.823} C_DIS
LIN {X -0.062,Y -537.007,Z 1210.934,A 0.000,B 0.000,C 90.000,E1 24.131} C_DIS
LIN {X 0.218,Y -530.772,Z 1210.930,A 0.000,B 0.000,C 90.000,E1 23.387} C_DIS
LIN {X -0.067,Y -524.461,Z 1210.926,A 0.000,B 0.000,C 90.000,E1 22.717} C_DIS
LIN {X 0.052,Y -513.757,Z 1210.920,A 0.000,B 0.000,C 90.000,E1 21.589} C_DIS
LIN {X -0.115,Y -504.333,Z 1210.915,A 0.000,B 0.000,C 90.000,E1 20.663} C_DIS
LIN {X 0.093,Y -494.464,Z 1210.910,A 0.000,B 0.000,C 90.000,E1 19.704} C_DIS
LIN {X 0.134,Y -485.851,Z 1210.905,A 0.000,B 0.000,C 90.000,E1 18.906} C_DIS
LIN {X 0.078,Y -474.206,Z 1210.899,A 0.000,B 0.000,C 90.000,E1 17.873} C_DIS
LIN {X -0.144,Y -461.009,Z 1210.893,A 0.000,B 0.000,C 90.000,E1 16.732} C_DIS
LIN {X -0.052,Y -437.658,Z 1210.881,A 0.000,B 0.000,C 90.000,E1 14.537} C_DIS
LIN {X -0.173,Y -421.945,Z 1210.872,A 0.000,B 0.000,C 90.000,E1 12.939} C_DIS
LIN {X -0.012,Y -405.214,Z 1210.861,A 0.000,B 0.000,C 90.000,E1 11.007} C_DIS
LIN {X 0.117,Y -397.741,Z 1210.856,A 0.000,B 0.000,C 90.000,E1 10.018} C_DIS
LIN {X 0.122,Y -396.617,Z 1210.855,A 0.000,B 0.000,C 90.000,E1 9.849} C_DIS
LIN {X -0.219,Y -394.465,Z 1210.853,A 0.000,B 0.000,C 90.000,E1 9.500} C_DIS
LIN {X 0.017,Y -394.114,Z 1210.852,A 0.000,B 0.000,C 90.000,E1 9.378} C_DIS
LIN {X 0.025,Y -393.484,Z 1210.851,A 0.000,B 0.000,C 90.000,E1 9.095} C_DIS
LIN {X -0.012,Y -393.482,Z 1210.851,A 0.000,B 0.000,C 90.000,E1 9.095} C_DIS
LIN {X -0.050,Y -394.030,Z 1210.849,A 0.000,B 0.000,C 90.000,E1 8.746} C_DIS
LIN {X 0.032,Y -396.937,Z 1210.845,A 0.000,B 0.000,C 90.000,E1 8.049} C_DIS
LIN {X -0.158,Y -401.147,Z 1210.842,A 0.000,B 0.000,C 90.000,E1 7.530} C_DIS
LIN {X -0.014,Y -406.623,Z 1210.839,A 0.000,B 0.000,C 90.000,E1 7.004} C_DIS
LIN {X -0.087,Y -425.994,Z 1210.831,A 0.000,B 0.000,C 90.000,E1 5.511} C_DIS
LIN {X 0.025,Y -437.157,Z 1210.826,A 0.000,B 0.000,C 90.000,E1 4.645} C_DIS
LIN {X 0.137,Y -452.896,Z 1210.819,A 0.000,B 0.000,C 90.000,E1 3.440} C_DIS
LIN {X 0.020,Y -462.266,Z 1210.815,A 0.000,B 0.000,C 90.000,E1 2.751} C_DIS
LIN {X -0.168,Y -469.981,Z 1210.812,A 0.000,B 0.000,C 90.000,E1 2.178} C_DIS
LIN {X 0.003,Y -477.524,Z 1210.809,A 0.000,B 0.000,C 90.000,E1 1.547} C_DIS
LIN {X 0.163,Y -484.563,Z 1210.805,A 0.000,B 0.000,C 90.000,E1 0.917} C_DIS
LIN {X -0.188,Y -491.610,Z 1210.802,A 0.000,B 0.000,C 90.000,E1 0.286} C_DIS
LIN {X -0.040,Y -497.597,Z 1210.798,A 0.000,B 0.000,C 90.000,E1 359.656} C_DIS
LIN {X -0.080,Y -505.252,Z 1210.793,A 0.000,B 0.000,C 90.000,E1 358.797} C_DIS
LIN {X 0.056,Y -511.154,Z 1210.789,A 0.000,B 0.000,C 90.000,E1 358.051} C_DIS
LIN {X 0.104,Y -516.737,Z 1210.785,A 0.000,B 0.000,C 90.000,E1 357.306} C_DIS
LIN {X -0.004,Y -520.909,Z 1210.782,A 0.000,B 0.000,C 90.000,E1 356.731} C_DIS
LIN {X 0.124,Y -525.674,Z 1210.778,A 0.000,B 0.000,C 90.000,E1 355.988} C_DIS
LIN {X -0.198,Y -529.974,Z 1210.774,A 0.000,B 0.000,C 90.000,E1 355.298} C_DIS
LIN {X -0.208,Y -533.166,Z 1210.771,A 0.000,B 0.000,C 90.000,E1 354.723} C_DIS
LIN {X 0.120,Y -536.783,Z 1210.767,A 0.000,B 0.000,C 90.000,E1 353.970} C_DIS
LIN {X -0.103,Y -540.037,Z 1210.763,A 0.000,B 0.000,C 90.000,E1 353.280} C_DIS
LIN {X 0.230,Y -543.012,Z 1210.759,A 0.000,B 0.000,C 90.000,E1 352.534} C_DIS
LIN {X -0.155,Y -545.205,Z 1210.756,A 0.000,B 0.000,C 90.000,E1 352.008} C_DIS
LIN {X 0.034,Y -548.197,Z 1210.751,A 0.000,B 0.000,C 90.000,E1 351.141} C_DIS
LIN {X 0.146,Y -550.009,Z 1210.748,A 0.000,B 0.000,C 90.000,E1 350.566} C_DIS
LIN {X 0.048,Y -553.382,Z 1210.741,A 0.000,B 0.000,C 90.000,E1 349.454} C_DIS
LIN {X -0.124,Y -555.667,Z 1210.737,A 0.000,B 0.000,C 90.000,E1 348.634} C_DIS
LIN {X 0.010,Y -559.242,Z 1210.729,A 0.000,B 0.000,C 90.000,E1 347.229} C_DIS
LIN {X 0.195,Y -562.328,Z 1210.721,A 0.000,B 0.000,C 90.000,E1 345.825} C_DIS
LIN {X 0.167,Y -565.136,Z 1210.714,A 0.000,B 0.000,C 90.000,E1 344.448} C_DIS
LIN {X -0.124,Y -567.267,Z 1210.708,A 0.000,B 0.000,C 90.000,E1 343.378} C_DIS
LIN {X -0.057,Y -569.592,Z 1210.700,A 0.000,B 0.000,C 90.000,E1 342.000} C_DIS
LIN {X 0.070,Y -570.864,Z 1210.695,A 0.000,B 0.000,C 90.000,E1 341.167} C_DIS
LIN {X 0.206,Y -572.274,Z 1210.689,A 0.000,B 0.000,C 90.000,E1 340.061} C_DIS
LIN {X 0.011,Y -573.179,Z 1210.685,A 0.000,B 0.000,C 90.000,E1 339.263} C_DIS
LIN {X -0.175,Y -573.904,Z 1210.680,A 0.000,B 0.000,C 90.000,E1 338.465} C_DIS
LIN {X 0.175,Y -574.323,Z 1210.676,A 0.000,B 0.000,C 90.000,E1 337.614} C_DIS
LIN {X 0.218,Y -574.449,Z 1210.671,A 0.000,B 0.000,C 90.000,E1 336.794} C_DIS
LIN {X -0.101,Y -574.425,Z 1210.668,A 0.000,B 0.000,C 90.000,E1 336.282} C_DIS
LIN {X -0.285,Y -573.998,Z 1210.664,A 0.000,B 0.000,C 90.000,E1 335.485} C_DIS
LIN {X -0.242,Y -573.365,Z 1210.659,A 0.000,B 0.000,C 90.000,E1 334.665} C_DIS
LIN {X 0.045,Y -572.209,Z 1210.655,A 0.000,B 0.000,C 90.000,E1 333.819} C_DIS
LIN {X 0.232,Y -571.253,Z 1210.652,A 0.000,B 0.000,C 90.000,E1 333.256} C_DIS
LIN {X -0.267,Y -569.444,Z 1210.647,A 0.000,B 0.000,C 90.000,E1 332.487} C_DIS
LIN {X -0.017,Y -567.384,Z 1210.642,A 0.000,B 0.000,C 90.000,E1 331.641} C_DIS
LIN {X 0.209,Y -564.904,Z 1210.638,A 0.000,B 0.000,C 90.000,E1 330.795} C_DIS
LIN {X 0.022,Y -563.908,Z 1210.636,A 0.000,B 0.000,C 90.000,E1 330.539} C_DIS
LIN {X -0.083,Y -561.673,Z 1210.633,A 0.000,B 0.000,C 90.000,E1 329.999} C_DIS
LIN {X -0.099,Y -559.723,Z 1210.631,A 0.000,B 0.000,C 90.000,E1 329.587} C_DIS
LIN {X 0.249,Y -556.829,Z 1210.628,A 0.000,B 0.000,C 90.000,E1 328.997} C_DIS
LIN {X 0.097,Y -553.577,Z 1210.625,A 0.000,B 0.000,C 90.000,E1 328.456} C_DIS
LIN {X -0.195,Y -548.928,Z 1210.621,A 0.000,B 0.000,C 90.000,E1 327.788} C_DIS
LIN {X 0.093,Y -542.858,Z 1210.616,A 0.000,B 0.000,C 90.000,E1 326.914} C_DIS
LIN {X 0.000,Y -537.260,Z 1210.612,A 0.000,B 0.000,C 90.000,E1 326.215} C_DIS
LIN {X -0.186,Y -530.301,Z 1210.608,A 0.000,B 0.000,C 90.000,E1 325.388} C_DIS
LIN {X -0.031,Y -519.618,Z 1210.600,A 0.000,B 0.000,C 90.000,E1 324.069} C_DIS
LIN {X -0.306,Y -516.746,Z 1210.598,A 0.000,B 0.000,C 90.000,E1 323.703} C_DIS
LIN {X 0.164,Y -513.611,Z 1210.595,A 0.000,B 0.000,C 90.000,E1 323.130} C_DIS
LIN {X -0.061,Y -511.578,Z 1210.593,A 0.000,B 0.000,C 90.000,E1 322.683} C_DIS
LIN {X -0.254,Y -511.083,Z 1210.592,A 0.000,B 0.000,C 90.000,E1 322.557} C_DIS
LIN {X -0.150,Y -510.120,Z 1210.589,A 0.000,B 0.000,C 90.000,E1 322.065} C_DIS
LIN {X 0.078,Y -509.680,Z 1210.588,A 0.000,B 0.000,C 90.000,E1 321.743} C_DIS
LIN {X -0.191,Y -509.399,Z 1210.583,A 0.000,B 0.000,C 90.000,E1 320.884} C_DIS
LIN {X 0.058,Y -510.968,Z 1210.564,A 0.000,B 0.000,C 90.000,E1 317.595} C_DIS
LIN {X 0.039,Y -512.191,Z 1210.553,A 0.000,B 0.000,C 90.000,E1 315.526} C_DIS
LIN {X 0.234,Y -512.967,Z 1210.545,A 0.000,B 0.000,C 90.000,E1 314.028} C_DIS
LIN {X -0.016,Y -513.929,Z 1210.535,A 0.000,B 0.000,C 90.000,E1 312.285} C_DIS
LIN {X -0.211,Y -514.861,Z 1210.525,A 0.000,B 0.000,C 90.000,E1 310.539} C_DIS
LIN {X -0.177,Y -515.479,Z 1210.519,A 0.000,B 0.000,C 90.000,E1 309.358} C_DIS
LIN {X -0.199,Y -516.123,Z 1210.510,A 0.000,B 0.000,C 90.000,E1 307.890} C_DIS
LIN {X 0.132,Y -516.771,Z 1210.501,A 0.000,B 0.000,C 90.000,E1 306.091} C_DIS
LIN {X 0.168,Y -517.602,Z 1210.491,A 0.000,B 0.000,C 90.000,E1 304.326} C_DIS
LIN {X -0.015,Y -518.166,Z 1210.483,A 0.000,B 0.000,C 90.000,E1 302.880} C_DIS
LIN {X -0.125,Y -518.592,Z 1210.476,A 0.000,B 0.000,C 90.000,E1 301.720} C_DIS
LIN {X 0.280,Y -518.825,Z 1210.471,A 0.000,B 0.000,C 90.000,E1 300.797} C_DIS
LIN {X 0.283,Y -519.070,Z 1210.463,A 0.000,B 0.000,C 90.000,E1 299.333} C_DIS
LIN {X 0.033,Y -519.287,Z 1210.455,A 0.000,B 0.000,C 90.000,E1 297.897} C_DIS
LIN {X -0.088,Y -519.428,Z 1210.445,A 0.000,B 0.000,C 90.000,E1 296.155} C_DIS
LIN {X -0.109,Y -519.463,Z 1210.437,A 0.000,B 0.000,C 90.000,E1 294.695} C_DIS
LIN {X -0.057,Y -519.517,Z 1210.426,A 0.000,B 0.000,C 90.000,E1 292.642} C_DIS
LIN {X -0.103,Y -519.596,Z 1210.421,A 0.000,B 0.000,C 90.000,E1 291.770} C_DIS
LIN {X 0.148,Y -519.452,Z 1210.416,A 0.000,B 0.000,C 90.000,E1 290.865} C_DIS
LIN {X 0.206,Y -519.054,Z 1210.408,A 0.000,B 0.000,C 90.000,E1 289.396} C_DIS
LIN {X 0.108,Y -518.501,Z 1210.401,A 0.000,B 0.000,C 90.000,E1 288.236} C_DIS
LIN {X -0.059,Y -517.566,Z 1210.392,A 0.000,B 0.000,C 90.000,E1 286.496} C_DIS
LIN {X 0.127,Y -516.616,Z 1210.384,A 0.000,B 0.000,C 90.000,E1 285.009} C_DIS
LIN {X 0.185,Y -515.875,Z 1210.377,A 0.000,B 0.000,C 90.000,E1 283.828} C_DIS
LIN {X 0.229,Y -515.154,Z 1210.370,A 0.000,B 0.000,C 90.000,E1 282.647} C_DIS
LIN {X 0.129,Y -514.188,Z 1210.362,A 0.000,B 0.000,C 90.000,E1 281.186} C_DIS
LIN {X -0.128,Y -512.979,Z 1210.351,A 0.000,B 0.000,C 90.000,E1 279.151} C_DIS
LIN {X -0.021,Y -511.534,Z 1210.338,A 0.000,B 0.000,C 90.000,E1 276.777} C_DIS
LIN {X 0.064,Y -510.489,Z 1210.328,A 0.000,B 0.000,C 90.000,E1 274.992} C_DIS
LIN {X -0.233,Y -509.790,Z 1210.321,A 0.000,B 0.000,C 90.000,E1 273.841} C_DIS
LIN {X 0.082,Y -508.393,Z 1210.308,A 0.000,B 0.000,C 90.000,E1 271.432} C_DIS
LIN {X 0.020,Y -507.455,Z 1210.298,A 0.000,B 0.000,C 90.000,E1 269.656} C_DIS
LIN {X 0.050,Y -506.594,Z 1210.290,A 0.000,B 0.000,C 90.000,E1 268.165} C_DIS
LIN {X 0.068,Y -505.665,Z 1210.282,A 0.000,B 0.000,C 90.000,E1 266.674} C_DIS
LIN {X 0.097,Y -504.655,Z 1210.273,A 0.000,B 0.000,C 90.000,E1 265.179} C_DIS
LIN {X 0.102,Y -503.525,Z 1210.265,A 0.000,B 0.000,C 90.000,E1 263.685} C_DIS
LIN {X 0.060,Y -501.754,Z 1210.255,A 0.000,B 0.000,C 90.000,E1 261.894} C_DIS
LIN {X 0.053,Y -500.252,Z 1210.245,A 0.000,B 0.000,C 90.000,E1 260.095} C_DIS
LIN {X 0.102,Y -498.789,Z 1210.235,A 0.000,B 0.000,C 90.000,E1 258.285} C_DIS
LIN {X 0.221,Y -497.398,Z 1210.225,A 0.000,B 0.000,C 90.000,E1 256.464} C_DIS
LIN {X -0.241,Y -495.663,Z 1210.212,A 0.000,B 0.000,C 90.000,E1 254.102} C_DIS
LIN {X 0.112,Y -494.824,Z 1210.205,A 0.000,B 0.000,C 90.000,E1 252.851} C_DIS
LIN {X 0.129,Y -494.191,Z 1210.198,A 0.000,B 0.000,C 90.000,E1 251.638} C_DIS
LIN {X 0.021,Y -493.401,Z 1210.190,A 0.000,B 0.000,C 90.000,E1 250.134} C_DIS
LIN {X 0.231,Y -492.382,Z 1210.181,A 0.000,B 0.000,C 90.000,E1 248.592} C_DIS
LIN {X -0.028,Y -491.224,Z 1210.173,A 0.000,B 0.000,C 90.000,E1 247.102} C_DIS
LIN {X -0.312,Y -489.723,Z 1210.164,A 0.000,B 0.000,C 90.000,E1 245.613} C_DIS
LIN {X -0.008,Y -488.439,Z 1210.158,A 0.000,B 0.000,C 90.000,E1 244.357} C_DIS
LIN {X 0.059,Y -486.798,Z 1210.149,A 0.000,B 0.000,C 90.000,E1 242.820} C_DIS
LIN {X -0.101,Y -483.509,Z 1210.134,A 0.000,B 0.000,C 90.000,E1 240.078} C_DIS
LIN {X -0.080,Y -481.606,Z 1210.125,A 0.000,B 0.000,C 90.000,E1 238.535} C_DIS
LIN {X -0.092,Y -478.972,Z 1210.113,A 0.000,B 0.000,C 90.000,E1 236.373} C_DIS
LIN {X 0.163,Y -476.780,Z 1210.103,A 0.000,B 0.000,C 90.000,E1 234.482} C_DIS
LIN {X 0.191,Y -475.047,Z 1210.094,A 0.000,B 0.000,C 90.000,E1 232.924} C_DIS
LIN {X -0.116,Y -472.992,Z 1210.084,A 0.000,B 0.000,C 90.000,E1 231.090} C_DIS
LIN {X -0.245,Y -471.337,Z 1210.075,A 0.000,B 0.000,C 90.000,E1 229.542} C_DIS
LIN {X -0.028,Y -469.437,Z 1210.065,A 0.000,B 0.000,C 90.000,E1 227.634} C_DIS
LIN {X 0.005,Y -466.737,Z 1210.049,A 0.000,B 0.000,C 90.000,E1 224.798} C_DIS
LIN {X -0.053,Y -464.711,Z 1210.033,A 0.000,B 0.000,C 90.000,E1 221.962} C_DIS
LIN {X -0.173,Y -464.117,Z 1210.012,A 0.000,B 0.000,C 90.000,E1 218.177} C_DIS
LIN {X 0.065,Y -464.708,Z 1210.000,A 0.000,B 0.000,C 90.000,E1 215.931} C_DIS
LIN {X 0.041,Y -465.790,Z 1209.984,A 0.000,B 0.000,C 90.000,E1 213.086} C_DIS
LIN {X -0.199,Y -467.968,Z 1209.970,A 0.000,B 0.000,C 90.000,E1 210.590} C_DIS
LIN {X -0.114,Y -471.357,Z 1209.952,A 0.000,B 0.000,C 90.000,E1 207.436} C_DIS
LIN {X 0.196,Y -474.029,Z 1209.940,A 0.000,B 0.000,C 90.000,E1 205.207} C_DIS
LIN {X 0.101,Y -480.669,Z 1209.916,A 0.000,B 0.000,C 90.000,E1 200.865} C_DIS
LIN {X 0.158,Y -489.239,Z 1209.894,A 0.000,B 0.000,C 90.000,E1 196.858} C_DIS
END
